// TIA Portal project "bary_callebaut" (V14)

(* hardware
DEVICE "S7-1200 station_1"  S7-1200 Station
   slot 0: "Rack_0"  S7-1200 Rack  Rack  V1.0
   slot 1: "PLC_1"  CPU 1214C DC/DC/DC  6ES7 214-1AG40-0XB0  V4.2
   slot 2: "DI 8/DQ 8x24VDC_1"  6ES7 223-1BH32-0XB0  V2.0
   slot 3: "SIWAREX WP231"  SIWAREX WP231  7MH4960-2AA01
DEVICE "GSD device_2"  GSD.Device.PN
   slot 0: "Rack"  Rack  V1.0
   slot 0: "danfoss-fc-series"  Danfoss FC PN  132B0348  V03.01.0
      slot 0: "Danfoss FC PN"  Danfoss FC PN
      slot 1: "Interface"  Interface
         slot 1: "Port 1"  Port 1
         slot 2: "Port 2"  Port 2
   slot 1: "PPO 6 - 4/4 Words, Danfoss Telegram 106_1"  PPO 6 - 4/4 Words, Danfoss Telegram 106
      slot 0: "Parameter Access Point"  Parameter Access Point
      slot 1: "PPO 6 - 4/4 Words, Danfoss Telegram 106"  PPO 6 - 4/4 Words, Danfoss Telegram 106
DEVICE "HMI"  TP700 Comfort
   slot 0: "HMI"  HMI  6AV2 124-0GC01-0AX0  13.0.1.0
   slot 1: "HMI_RT_2"  TP700 Comfort  6AV2 124-0GC01-0AX0  13.0.1.0
   slot 5: "HMI.IE_CP_1"  PROFINET Schnittstelle
      slot 1: "PROFINET Schnittstelle_1"  PROFINET Schnittstelle
         slot 1: "Port_1"  Port
         slot 2: "Port_2"  Port
   slot 7: "HMI.MPI/DP_CP_1"  MPI/DP Schnittstelle
DEVICE "HMI_1"  KTP700 Basic PN
   slot 0: "KTP700 Basic PN"  KTP700 Basic PN  6AV2 123-2GB03-0AX0  14.0.1.0
   slot 1: "HMI_RT_1"  KTP700 Basic PN  6AV2 123-2GB03-0AX0  14.0.1.0
   slot 5: "HMI_1.IE_CP_1"  PROFINET Interface  14.0.1.0
      slot 1: "PROFINET Interface_1"  PROFINET Interface
         slot 1: "Port_1"  Port
*)

// ===== PLC "PLC_1"  CPU 1214C DC/DC/DC =====
// protected blocks, not shown: "WP231PR"

VAR_GLOBAL   // PLC tag table "Default tag table"
   "Voltage_CPU_Ok" AT %I0.0 : Bool;   // Питание контрллера в номе
   "Voltage_DI_Ok" AT %I0.1 : Bool;   // Питание DI в норме
   "Voltage_DO_Ok" AT %I0.2 : Bool;   // Питание DO в норме
   "Voltage_24V_Ok" AT %I0.3 : Bool;   // Питание 24В в норме
   "Safety_Ok" AT %I0.4 : Bool;   // Безопасность в норме
   "Cold_tunnel_QF" AT %I0.5 : Bool;   // Защитный автомат холодный тунель
   "T1_QF" AT %I0.6 : Bool;   // Защитный автомат Т1
   "T2_QF" AT %I0.7 : Bool;   // Защитный автомат Т2
   "T3_QF" AT %I1.0 : Bool;   // Защитный автомат Т3
   "T2_Box_ready" AT %I1.1 : Bool;   // Датчик наличия коробки
   "T3_Box_ready" AT %I1.2 : Bool;   // Датчик наличия коробки
   "T4_Box_ready" AT %I1.3 : Bool;   // Датчик наличия коробки
   "Air_pressure_Ok" AT %I1.4 : Bool;   // Давление воздуха
   "FB_K1_Close" AT %I2.0 : Bool;   // Закрыто
   "FB_K2_Open" AT %I2.1 : Bool;   // Открыто
   "FB_K2_Close" AT %I2.2 : Bool;   // Закрыто
   "FB_K3_Open" AT %I2.3 : Bool;   // Открыто
   "FB_K3_Close" AT %I2.4 : Bool;   // Закрыто
   "T0_CMD" AT %Q0.0 : Bool;   // Вкл Т0
   "T1_CMD" AT %Q0.1 : Bool;   // Вкл Т1
   "T2_CMD" AT %Q0.2 : Bool;   // Вкл Т2
   "T3_CMD" AT %Q0.3 : Bool;   // Вкл Т3
   "K1_CMD" AT %Q0.4 : Bool;   // Вкл/выкл К1
   "K2_CMD" AT %Q0.5 : Bool;   // Вкл К2
   "K3_CMD" AT %Q0.6 : Bool;   // Вкл К3
   "Supply_allowed" AT %Q0.7 : Bool;   // Подача шоколада разрешена (отдаем другой системе)
   "Reset_safety" AT %Q2.0 : Bool;   // Сброс безопасности
   "Reset" AT %Q2.1 : Bool;   // Сброс
   "Green" AT %Q2.4 : Bool;   // Зеленый
   "Red" AT %Q2.5 : Bool;   // Красный
   "Blue" AT %Q2.6 : Bool;   // Синий
   "Orange" AT %Q2.7 : Bool;   // Оранжевый
   "Tag_1" AT %MW50 : Int;
   "Tag_2" AT %M100.0 : Bool;
END_VAR

VAR_GLOBAL   // PLC tag table "CF_tegs"
   "Status_word_input" AT %IW50 : Int;
   "MAV_input" AT %IW52 : Int;
   "Motor_torque_input" AT %IW54 : Int;
   "Digital_input" AT %IW56 : Int;
   "Control_word_output" AT %QW50 : Int;
   "Not_used_output" AT %QW54 : Int;
   "Reference_output" AT %QW52 : Int;
   "Not_used_output(1)" AT %QW56 : Int;
END_VAR

VAR_GLOBAL   // PLC tag table "Sys"
   "ON" AT %M2.0 : Bool;
   "OFF" AT %M2.1 : Bool;
   "pulse_01s" AT %M3.0 : Bool;
   "pulse_05s" AT %M3.1 : Bool;
   "pulse_1s" AT %M3.2 : Bool;
   "pulse_1m" AT %M3.3 : Bool;
   "pulse_1h" AT %M3.4 : Bool;
   "All_block" AT %M4.0 : Bool;
   "Reset_All" AT %M4.1 : Bool;
   "Sim_All" AT %M4.2 : Bool;
   "Global_Alm" AT %M4.3 : Bool;
   "ToAuto" AT %M4.4 : Bool;
   "ToHand" AT %M4.5 : Bool;
   "Any_Hand" AT %M5.0 : Bool;
   "DI_Hand" AT %M5.1 : Bool;
   "DO_Hand" AT %M5.2 : Bool;
   "AI_Hand" AT %M5.3 : Bool;
   "AO_Hand" AT %M5.4 : Bool;
   "M_Hand" AT %M5.5 : Bool;
   "V_Hand" AT %M5.6 : Bool;
   "X_Hand" AT %M5.7 : Bool;
   "System_Byte" AT %MB1 : Byte;
   "FirstScan" AT %M1.0 : Bool;
   "DiagStatusUpdate" AT %M1.1 : Bool;
   "AlwaysTRUE" AT %M1.2 : Bool;
   "AlwaysFALSE" AT %M1.3 : Bool;
   "Clock_Byte" AT %MB0 : Byte;
   "Clock_10Hz" AT %M0.0 : Bool;
   "Clock_5Hz" AT %M0.1 : Bool;
   "Clock_2.5Hz" AT %M0.2 : Bool;
   "Clock_2Hz" AT %M0.3 : Bool;
   "Clock_1.25Hz" AT %M0.4 : Bool;
   "Clock_1Hz" AT %M0.5 : Bool;
   "Clock_0.625Hz" AT %M0.6 : Bool;
   "Clock_0.5Hz" AT %M0.7 : Bool;
   "DI_Alm" AT %M6.0 : Bool;
   "DO_Alm" AT %M6.1 : Bool;
   "AI_Alm" AT %M6.2 : Bool;
   "AO_Alm" AT %M6.3 : Bool;
   "M_Alm" AT %M6.4 : Bool;
   "V_Alm" AT %M6.5 : Bool;
   "X_Alm" AT %M6.6 : Bool;
   "Any_Alm" AT %M6.7 : Bool;
   "W_Alm" AT %M7.0 : Bool;
   "RPD_Alm" AT %M7.1 : Bool;
   "I_Alm" AT %M7.2 : Bool;
   "O1_Alm" AT %M7.3 : Bool;
   "O2_Alm" AT %M7.4 : Bool;
   "VT_Alm" AT %M7.5 : Bool;
   "FStop" AT %M7.6 : Bool;
   "pulse_5s" AT %M3.5 : Bool;
   "Clock_5s" AT %M3.6 : Bool;
   "pos_1s" AT %M8.0 : Bool;
   "pos_05s" AT %M8.1 : Bool;
   "pos_01s" AT %M8.2 : Bool;
   "neg_01s" AT %M8.3 : Bool;
END_VAR

DATA_BLOCK "Logic_DB"   // DB4
{ S7_Optimized_Access := 'FALSE' }
VERSION : 0.1
// stored: InstanceOfName Logic
"Logic"
BEGIN
   T_reset_mem.SP := 10.0;
END_DATA_BLOCK

DATA_BLOCK "T4D4_DB"   // DB10
{ S7_Optimized_Access := 'FALSE' }
VERSION : 0.1
// stored: InstanceOfName T4D4
"T4D4"
BEGIN
   S2.One := 0.1;
   S2.SP := 5.0;
   S1.One := 0.1;
   S1.SP := 2.0;
END_DATA_BLOCK

DATA_BLOCK "T3V3W3_DB"   // DB11
{ S7_Optimized_Access := 'FALSE' }
VERSION : 0.1
// stored: InstanceOfName T3V3W3
"T3V3W3"
BEGIN
END_DATA_BLOCK

DATA_BLOCK "T2D2_DB"   // DB12
{ S7_Optimized_Access := 'FALSE' }
VERSION : 0.1
// stored: InstanceOfName T2D2
"T2D2"
BEGIN
END_DATA_BLOCK

DATA_BLOCK "T0T1_DB"   // DB13
{ S7_Optimized_Access := 'FALSE' }
VERSION : 0.1
// stored: InstanceOfName T0T1
"T0T1"
BEGIN
END_DATA_BLOCK

DATA_BLOCK "del_stat_mem_DB"   // DB14
{ S7_Optimized_Access := 'FALSE' }
VERSION : 0.1
// stored: InstanceOfName del_stat_mem
"del_stat_mem"
BEGIN
END_DATA_BLOCK

DATA_BLOCK "move_pn_DB"   // DB16
{ S7_Optimized_Access := 'FALSE' }
VERSION : 0.1
// stored: InstanceOfName move_pn
"move_pn"
BEGIN
END_DATA_BLOCK

DATA_BLOCK "Reset_st_DB"   // DB17
{ S7_Optimized_Access := 'FALSE' }
VERSION : 0.1
// stored: InstanceOfName Reset_st
"Reset_st"
BEGIN
END_DATA_BLOCK

DATA_BLOCK "Statistic_DB"   // DB19
{ S7_Optimized_Access := 'FALSE' }
VERSION : 0.1
// stored: InstanceOfName Statistic
"Statistic"
BEGIN
END_DATA_BLOCK

DATA_BLOCK "prepare_DB"   // DB20
{ S7_Optimized_Access := 'TRUE' }
VERSION : 0.1
// stored: InstanceOfName prepare
"prepare"
BEGIN
END_DATA_BLOCK

// folder: Modules

DATA_BLOCK "Profinet_FC280_DB"   // DB1
{ S7_Optimized_Access := 'FALSE' }
VERSION : 0.1
// stored: InstanceOfName Profinet_FC280
"Profinet_FC280"
BEGIN
END_DATA_BLOCK

DATA_BLOCK "Motors_DB"   // DB2
{ S7_Optimized_Access := 'FALSE' }
VERSION : 0.1
// stored: InstanceOfName Motors
"Motors"
BEGIN
END_DATA_BLOCK

DATA_BLOCK "Valves_DB"   // DB3
{ S7_Optimized_Access := 'FALSE' }
VERSION : 0.1
// stored: InstanceOfName Valves
"Valves"
BEGIN
END_DATA_BLOCK

DATA_BLOCK "DRV_CF_DB"   // DB5
{ S7_Optimized_Access := 'FALSE' }
VERSION : 0.1
// stored: InstanceOfName DRV_CF
"DRV_CF"
BEGIN
END_DATA_BLOCK

DATA_BLOCK "DOx_DB"   // DB6
{ S7_Optimized_Access := 'FALSE' }
VERSION : 0.1
// stored: InstanceOfName DOx
"DOx"
BEGIN
END_DATA_BLOCK

DATA_BLOCK "AOx_DB"   // DB8
{ S7_Optimized_Access := 'FALSE' }
VERSION : 0.1
// stored: InstanceOfName AOx
"AOx"
BEGIN
END_DATA_BLOCK

DATA_BLOCK "DIx_DB"   // DB9
{ S7_Optimized_Access := 'FALSE' }
VERSION : 0.1
// stored: InstanceOfName DIx
"DIx"
BEGIN
END_DATA_BLOCK

// folder: System blocks/Program resources

DATA_BLOCK "T_Reset"   // DB7
{ S7_Optimized_Access := 'TRUE' }
AUTHOR : Simatic
FAMILY : IEC
NAME : IEC_TMR
VERSION : 1.0
// stored: InstanceOfName IEC_TIMER
"IEC_TIMER"
BEGIN
END_DATA_BLOCK

DATA_BLOCK "clock_5s_ON"   // DB507
{ S7_Optimized_Access := 'TRUE' }
AUTHOR : Simatic
FAMILY : IEC
NAME : IEC_TMR
VERSION : 1.0
// stored: InstanceOfName IEC_TIMER
"IEC_TIMER"
BEGIN
END_DATA_BLOCK

DATA_BLOCK "clock_5s_OFF"   // DB508
{ S7_Optimized_Access := 'TRUE' }
AUTHOR : Simatic
FAMILY : IEC
NAME : IEC_TMR
VERSION : 1.0
// stored: InstanceOfName IEC_TIMER
"IEC_TIMER"
BEGIN
END_DATA_BLOCK

// folder: db_flash

DATA_BLOCK "data"   // DB15
{ S7_Optimized_Access := 'FALSE' }
VERSION : 0.1
   VAR
      newName : String := 'newlog';
      "name" : String := 'log';
      logID : DWord;
      logHeader : String := 'count,weight';
      myData : Struct
         number : Int;
         weight : Real;
      END_STRUCT;
      executeCreate : Bool;
      crateDone : Bool;
      createBusy : Bool;
      createError : Bool;
      createStatus : Word;
      createStatusMem : Word;
      dlogCreated : Bool;
   END_VAR
BEGIN
END_DATA_BLOCK

DATA_BLOCK "logW"   // DB21
{ S7_Optimized_Access := 'TRUE' }
VERSION : 0.1
   VAR
      executeWrite : Bool;
      count : Int;
      scaledTemp : Real;
      scaledPressure : Real;
      writeDone : Bool;
      writeBusy : Bool;
      writeError : Bool;
      writeFullStatus : Word;
      closeDone : Bool;
      closeBusy : Bool;
      closeError : Bool;
      closeStatus : Word;
      executeOpen : Bool;
      openDone : Bool;
      openBusy : Bool;
      openError : Bool;
      openStatus : Word;
      executeNewFile : Bool;
      fileDone : Bool;
      fileBusy : Bool;
      fileError : Bool;
      fileStatus : Word;
   END_VAR
BEGIN
END_DATA_BLOCK

DATA_BLOCK "logFB"   // DB22
{ S7_Optimized_Access := 'TRUE' }
VERSION : 0.1
BEGIN
END_DATA_BLOCK

// folder: statistic

DATA_BLOCK "bd"   // DB18
{ S7_Optimized_Access := 'FALSE' }
VERSION : 0.1
   VAR
      weight_box : Array[1..3000] of Real;
   END_VAR
BEGIN
   weight_box[1] := 0.0;
   weight_box[2] := 0.0;
   weight_box[3] := 0.0;
   weight_box[4] := 0.0;
   weight_box[5] := 0.0;
   weight_box[6] := 0.0;
   weight_box[7] := 0.0;
   weight_box[8] := 0.0;
   weight_box[9] := 0.0;
   weight_box[10] := 0.0;
   weight_box[11] := 0.0;
   weight_box[12] := 0.0;
   weight_box[13] := 0.0;
   weight_box[14] := 0.0;
   weight_box[15] := 0.0;
   weight_box[16] := 0.0;
   weight_box[17] := 0.0;
   weight_box[18] := 0.0;
   weight_box[19] := 0.0;
   weight_box[20] := 0.0;
   weight_box[21] := 0.0;
   weight_box[22] := 0.0;
   weight_box[23] := 0.0;
   weight_box[24] := 0.0;
   weight_box[25] := 0.0;
   weight_box[26] := 0.0;
   weight_box[27] := 0.0;
   weight_box[28] := 0.0;
   weight_box[29] := 0.0;
   weight_box[30] := 0.0;
   weight_box[31] := 0.0;
   weight_box[32] := 0.0;
   weight_box[33] := 0.0;
   weight_box[34] := 0.0;
   weight_box[35] := 0.0;
   weight_box[36] := 0.0;
   weight_box[37] := 0.0;
   weight_box[38] := 0.0;
   weight_box[39] := 0.0;
   weight_box[40] := 0.0;
   weight_box[41] := 0.0;
   weight_box[42] := 0.0;
   weight_box[43] := 0.0;
   weight_box[44] := 0.0;
   weight_box[45] := 0.0;
   weight_box[46] := 0.0;
   weight_box[47] := 0.0;
   weight_box[48] := 0.0;
   weight_box[49] := 0.0;
   weight_box[50] := 0.0;
   weight_box[51] := 0.0;
   weight_box[52] := 0.0;
   weight_box[53] := 0.0;
   weight_box[54] := 0.0;
   weight_box[55] := 0.0;
   weight_box[56] := 0.0;
   weight_box[57] := 0.0;
   weight_box[58] := 0.0;
   weight_box[59] := 0.0;
   weight_box[60] := 0.0;
   weight_box[61] := 0.0;
   weight_box[62] := 0.0;
   weight_box[63] := 0.0;
   weight_box[64] := 0.0;
   weight_box[65] := 0.0;
   weight_box[66] := 0.0;
   weight_box[67] := 0.0;
   weight_box[68] := 0.0;
   weight_box[69] := 0.0;
   weight_box[70] := 0.0;
   weight_box[71] := 0.0;
   weight_box[72] := 0.0;
   weight_box[73] := 0.0;
   weight_box[74] := 0.0;
   weight_box[75] := 0.0;
   weight_box[76] := 0.0;
   weight_box[77] := 0.0;
   weight_box[78] := 0.0;
   weight_box[79] := 0.0;
   weight_box[80] := 0.0;
   weight_box[81] := 0.0;
   weight_box[82] := 0.0;
   weight_box[83] := 0.0;
   weight_box[84] := 0.0;
   weight_box[85] := 0.0;
   weight_box[86] := 0.0;
   weight_box[87] := 0.0;
   weight_box[88] := 0.0;
   weight_box[89] := 0.0;
   weight_box[90] := 0.0;
   weight_box[91] := 0.0;
   weight_box[92] := 0.0;
   weight_box[93] := 0.0;
   weight_box[94] := 0.0;
   weight_box[95] := 0.0;
   weight_box[96] := 0.0;
   weight_box[97] := 0.0;
   weight_box[98] := 0.0;
   weight_box[99] := 0.0;
   weight_box[100] := 0.0;
   weight_box[101] := 0.0;
   weight_box[102] := 0.0;
   weight_box[103] := 0.0;
   weight_box[104] := 0.0;
   weight_box[105] := 0.0;
   weight_box[106] := 0.0;
   weight_box[107] := 0.0;
   weight_box[108] := 0.0;
   weight_box[109] := 0.0;
   weight_box[110] := 0.0;
   weight_box[111] := 0.0;
   weight_box[112] := 0.0;
   weight_box[113] := 0.0;
   weight_box[114] := 0.0;
   weight_box[115] := 0.0;
   weight_box[116] := 0.0;
   weight_box[117] := 0.0;
   weight_box[118] := 0.0;
   weight_box[119] := 0.0;
   weight_box[120] := 0.0;
   weight_box[121] := 0.0;
   weight_box[122] := 0.0;
   weight_box[123] := 0.0;
   weight_box[124] := 0.0;
   weight_box[125] := 0.0;
   weight_box[126] := 0.0;
   weight_box[127] := 0.0;
   weight_box[128] := 0.0;
   weight_box[129] := 0.0;
   weight_box[130] := 0.0;
   weight_box[131] := 0.0;
   weight_box[132] := 0.0;
   weight_box[133] := 0.0;
   weight_box[134] := 0.0;
   weight_box[135] := 0.0;
   weight_box[136] := 0.0;
   weight_box[137] := 0.0;
   weight_box[138] := 0.0;
   weight_box[139] := 0.0;
   weight_box[140] := 0.0;
   weight_box[141] := 0.0;
   weight_box[142] := 0.0;
   weight_box[143] := 0.0;
   weight_box[144] := 0.0;
   weight_box[145] := 0.0;
   weight_box[146] := 0.0;
   weight_box[147] := 0.0;
   weight_box[148] := 0.0;
   weight_box[149] := 0.0;
   weight_box[150] := 0.0;
   weight_box[151] := 0.0;
   weight_box[152] := 0.0;
   weight_box[153] := 0.0;
   weight_box[154] := 0.0;
   weight_box[155] := 0.0;
   weight_box[156] := 0.0;
   weight_box[157] := 0.0;
   weight_box[158] := 0.0;
   weight_box[159] := 0.0;
   weight_box[160] := 0.0;
   weight_box[161] := 0.0;
   weight_box[162] := 0.0;
   weight_box[163] := 0.0;
   weight_box[164] := 0.0;
   weight_box[165] := 0.0;
   weight_box[166] := 0.0;
   weight_box[167] := 0.0;
   weight_box[168] := 0.0;
   weight_box[169] := 0.0;
   weight_box[170] := 0.0;
   weight_box[171] := 0.0;
   weight_box[172] := 0.0;
   weight_box[173] := 0.0;
   weight_box[174] := 0.0;
   weight_box[175] := 0.0;
   weight_box[176] := 0.0;
   weight_box[177] := 0.0;
   weight_box[178] := 0.0;
   weight_box[179] := 0.0;
   weight_box[180] := 0.0;
   weight_box[181] := 0.0;
   weight_box[182] := 0.0;
   weight_box[183] := 0.0;
   weight_box[184] := 0.0;
   weight_box[185] := 0.0;
   weight_box[186] := 0.0;
   weight_box[187] := 0.0;
   weight_box[188] := 0.0;
   weight_box[189] := 0.0;
   weight_box[190] := 0.0;
   weight_box[191] := 0.0;
   weight_box[192] := 0.0;
   weight_box[193] := 0.0;
   weight_box[194] := 0.0;
   weight_box[195] := 0.0;
   weight_box[196] := 0.0;
   weight_box[197] := 0.0;
   weight_box[198] := 0.0;
   weight_box[199] := 0.0;
   weight_box[200] := 0.0;
   weight_box[201] := 0.0;
   weight_box[202] := 0.0;
   weight_box[203] := 0.0;
   weight_box[204] := 0.0;
   weight_box[205] := 0.0;
   weight_box[206] := 0.0;
   weight_box[207] := 0.0;
   weight_box[208] := 0.0;
   weight_box[209] := 0.0;
   weight_box[210] := 0.0;
   weight_box[211] := 0.0;
   weight_box[212] := 0.0;
   weight_box[213] := 0.0;
   weight_box[214] := 0.0;
   weight_box[215] := 0.0;
   weight_box[216] := 0.0;
   weight_box[217] := 0.0;
   weight_box[218] := 0.0;
   weight_box[219] := 0.0;
   weight_box[220] := 0.0;
   weight_box[221] := 0.0;
   weight_box[222] := 0.0;
   weight_box[223] := 0.0;
   weight_box[224] := 0.0;
   weight_box[225] := 0.0;
   weight_box[226] := 0.0;
   weight_box[227] := 0.0;
   weight_box[228] := 0.0;
   weight_box[229] := 0.0;
   weight_box[230] := 0.0;
   weight_box[231] := 0.0;
   weight_box[232] := 0.0;
   weight_box[233] := 0.0;
   weight_box[234] := 0.0;
   weight_box[235] := 0.0;
   weight_box[236] := 0.0;
   weight_box[237] := 0.0;
   weight_box[238] := 0.0;
   weight_box[239] := 0.0;
   weight_box[240] := 0.0;
   weight_box[241] := 0.0;
   weight_box[242] := 0.0;
   weight_box[243] := 0.0;
   weight_box[244] := 0.0;
   weight_box[245] := 0.0;
   weight_box[246] := 0.0;
   weight_box[247] := 0.0;
   weight_box[248] := 0.0;
   weight_box[249] := 0.0;
   weight_box[250] := 0.0;
   weight_box[251] := 0.0;
   weight_box[252] := 0.0;
   weight_box[253] := 0.0;
   weight_box[254] := 0.0;
   weight_box[255] := 0.0;
   weight_box[256] := 0.0;
   weight_box[257] := 0.0;
   weight_box[258] := 0.0;
   weight_box[259] := 0.0;
   weight_box[260] := 0.0;
   weight_box[261] := 0.0;
   weight_box[262] := 0.0;
   weight_box[263] := 0.0;
   weight_box[264] := 0.0;
   weight_box[265] := 0.0;
   weight_box[266] := 0.0;
   weight_box[267] := 0.0;
   weight_box[268] := 0.0;
   weight_box[269] := 0.0;
   weight_box[270] := 0.0;
   weight_box[271] := 0.0;
   weight_box[272] := 0.0;
   weight_box[273] := 0.0;
   weight_box[274] := 0.0;
   weight_box[275] := 0.0;
   weight_box[276] := 0.0;
   weight_box[277] := 0.0;
   weight_box[278] := 0.0;
   weight_box[279] := 0.0;
   weight_box[280] := 0.0;
   weight_box[281] := 0.0;
   weight_box[282] := 0.0;
   weight_box[283] := 0.0;
   weight_box[284] := 0.0;
   weight_box[285] := 0.0;
   weight_box[286] := 0.0;
   weight_box[287] := 0.0;
   weight_box[288] := 0.0;
   weight_box[289] := 0.0;
   weight_box[290] := 0.0;
   weight_box[291] := 0.0;
   weight_box[292] := 0.0;
   weight_box[293] := 0.0;
   weight_box[294] := 0.0;
   weight_box[295] := 0.0;
   weight_box[296] := 0.0;
   weight_box[297] := 0.0;
   weight_box[298] := 0.0;
   weight_box[299] := 0.0;
   weight_box[300] := 0.0;
   weight_box[301] := 0.0;
   weight_box[302] := 0.0;
   weight_box[303] := 0.0;
   weight_box[304] := 0.0;
   weight_box[305] := 0.0;
   weight_box[306] := 0.0;
   weight_box[307] := 0.0;
   weight_box[308] := 0.0;
   weight_box[309] := 0.0;
   weight_box[310] := 0.0;
   weight_box[311] := 0.0;
   weight_box[312] := 0.0;
   weight_box[313] := 0.0;
   weight_box[314] := 0.0;
   weight_box[315] := 0.0;
   weight_box[316] := 0.0;
   weight_box[317] := 0.0;
   weight_box[318] := 0.0;
   weight_box[319] := 0.0;
   weight_box[320] := 0.0;
   weight_box[321] := 0.0;
   weight_box[322] := 0.0;
   weight_box[323] := 0.0;
   weight_box[324] := 0.0;
   weight_box[325] := 0.0;
   weight_box[326] := 0.0;
   weight_box[327] := 0.0;
   weight_box[328] := 0.0;
   weight_box[329] := 0.0;
   weight_box[330] := 0.0;
   weight_box[331] := 0.0;
   weight_box[332] := 0.0;
   weight_box[333] := 0.0;
   weight_box[334] := 0.0;
   weight_box[335] := 0.0;
   weight_box[336] := 0.0;
   weight_box[337] := 0.0;
   weight_box[338] := 0.0;
   weight_box[339] := 0.0;
   weight_box[340] := 0.0;
   weight_box[341] := 0.0;
   weight_box[342] := 0.0;
   weight_box[343] := 0.0;
   weight_box[344] := 0.0;
   weight_box[345] := 0.0;
   weight_box[346] := 0.0;
   weight_box[347] := 0.0;
   weight_box[348] := 0.0;
   weight_box[349] := 0.0;
   weight_box[350] := 0.0;
   weight_box[351] := 0.0;
   weight_box[352] := 0.0;
   weight_box[353] := 0.0;
   weight_box[354] := 0.0;
   weight_box[355] := 0.0;
   weight_box[356] := 0.0;
   weight_box[357] := 0.0;
   weight_box[358] := 0.0;
   weight_box[359] := 0.0;
   weight_box[360] := 0.0;
   weight_box[361] := 0.0;
   weight_box[362] := 0.0;
   weight_box[363] := 0.0;
   weight_box[364] := 0.0;
   weight_box[365] := 0.0;
   weight_box[366] := 0.0;
   weight_box[367] := 0.0;
   weight_box[368] := 0.0;
   weight_box[369] := 0.0;
   weight_box[370] := 0.0;
   weight_box[371] := 0.0;
   weight_box[372] := 0.0;
   weight_box[373] := 0.0;
   weight_box[374] := 0.0;
   weight_box[375] := 0.0;
   weight_box[376] := 0.0;
   weight_box[377] := 0.0;
   weight_box[378] := 0.0;
   weight_box[379] := 0.0;
   weight_box[380] := 0.0;
   weight_box[381] := 0.0;
   weight_box[382] := 0.0;
   weight_box[383] := 0.0;
   weight_box[384] := 0.0;
   weight_box[385] := 0.0;
   weight_box[386] := 0.0;
   weight_box[387] := 0.0;
   weight_box[388] := 0.0;
   weight_box[389] := 0.0;
   weight_box[390] := 0.0;
   weight_box[391] := 0.0;
   weight_box[392] := 0.0;
   weight_box[393] := 0.0;
   weight_box[394] := 0.0;
   weight_box[395] := 0.0;
   weight_box[396] := 0.0;
   weight_box[397] := 0.0;
   weight_box[398] := 0.0;
   weight_box[399] := 0.0;
   weight_box[400] := 0.0;
   weight_box[401] := 0.0;
   weight_box[402] := 0.0;
   weight_box[403] := 0.0;
   weight_box[404] := 0.0;
   weight_box[405] := 0.0;
   weight_box[406] := 0.0;
   weight_box[407] := 0.0;
   weight_box[408] := 0.0;
   weight_box[409] := 0.0;
   weight_box[410] := 0.0;
   weight_box[411] := 0.0;
   weight_box[412] := 0.0;
   weight_box[413] := 0.0;
   weight_box[414] := 0.0;
   weight_box[415] := 0.0;
   weight_box[416] := 0.0;
   weight_box[417] := 0.0;
   weight_box[418] := 0.0;
   weight_box[419] := 0.0;
   weight_box[420] := 0.0;
   weight_box[421] := 0.0;
   weight_box[422] := 0.0;
   weight_box[423] := 0.0;
   weight_box[424] := 0.0;
   weight_box[425] := 0.0;
   weight_box[426] := 0.0;
   weight_box[427] := 0.0;
   weight_box[428] := 0.0;
   weight_box[429] := 0.0;
   weight_box[430] := 0.0;
   weight_box[431] := 0.0;
   weight_box[432] := 0.0;
   weight_box[433] := 0.0;
   weight_box[434] := 0.0;
   weight_box[435] := 0.0;
   weight_box[436] := 0.0;
   weight_box[437] := 0.0;
   weight_box[438] := 0.0;
   weight_box[439] := 0.0;
   weight_box[440] := 0.0;
   weight_box[441] := 0.0;
   weight_box[442] := 0.0;
   weight_box[443] := 0.0;
   weight_box[444] := 0.0;
   weight_box[445] := 0.0;
   weight_box[446] := 0.0;
   weight_box[447] := 0.0;
   weight_box[448] := 0.0;
   weight_box[449] := 0.0;
   weight_box[450] := 0.0;
   weight_box[451] := 0.0;
   weight_box[452] := 0.0;
   weight_box[453] := 0.0;
   weight_box[454] := 0.0;
   weight_box[455] := 0.0;
   weight_box[456] := 0.0;
   weight_box[457] := 0.0;
   weight_box[458] := 0.0;
   weight_box[459] := 0.0;
   weight_box[460] := 0.0;
   weight_box[461] := 0.0;
   weight_box[462] := 0.0;
   weight_box[463] := 0.0;
   weight_box[464] := 0.0;
   weight_box[465] := 0.0;
   weight_box[466] := 0.0;
   weight_box[467] := 0.0;
   weight_box[468] := 0.0;
   weight_box[469] := 0.0;
   weight_box[470] := 0.0;
   weight_box[471] := 0.0;
   weight_box[472] := 0.0;
   weight_box[473] := 0.0;
   weight_box[474] := 0.0;
   weight_box[475] := 0.0;
   weight_box[476] := 0.0;
   weight_box[477] := 0.0;
   weight_box[478] := 0.0;
   weight_box[479] := 0.0;
   weight_box[480] := 0.0;
   weight_box[481] := 0.0;
   weight_box[482] := 0.0;
   weight_box[483] := 0.0;
   weight_box[484] := 0.0;
   weight_box[485] := 0.0;
   weight_box[486] := 0.0;
   weight_box[487] := 0.0;
   weight_box[488] := 0.0;
   weight_box[489] := 0.0;
   weight_box[490] := 0.0;
   weight_box[491] := 0.0;
   weight_box[492] := 0.0;
   weight_box[493] := 0.0;
   weight_box[494] := 0.0;
   weight_box[495] := 0.0;
   weight_box[496] := 0.0;
   weight_box[497] := 0.0;
   weight_box[498] := 0.0;
   weight_box[499] := 0.0;
   weight_box[500] := 0.0;
   weight_box[501] := 0.0;
   weight_box[502] := 0.0;
   weight_box[503] := 0.0;
   weight_box[504] := 0.0;
   weight_box[505] := 0.0;
   weight_box[506] := 0.0;
   weight_box[507] := 0.0;
   weight_box[508] := 0.0;
   weight_box[509] := 0.0;
   weight_box[510] := 0.0;
   weight_box[511] := 0.0;
   weight_box[512] := 0.0;
   weight_box[513] := 0.0;
   weight_box[514] := 0.0;
   weight_box[515] := 0.0;
   weight_box[516] := 0.0;
   weight_box[517] := 0.0;
   weight_box[518] := 0.0;
   weight_box[519] := 0.0;
   weight_box[520] := 0.0;
   weight_box[521] := 0.0;
   weight_box[522] := 0.0;
   weight_box[523] := 0.0;
   weight_box[524] := 0.0;
   weight_box[525] := 0.0;
   weight_box[526] := 0.0;
   weight_box[527] := 0.0;
   weight_box[528] := 0.0;
   weight_box[529] := 0.0;
   weight_box[530] := 0.0;
   weight_box[531] := 0.0;
   weight_box[532] := 0.0;
   weight_box[533] := 0.0;
   weight_box[534] := 0.0;
   weight_box[535] := 0.0;
   weight_box[536] := 0.0;
   weight_box[537] := 0.0;
   weight_box[538] := 0.0;
   weight_box[539] := 0.0;
   weight_box[540] := 0.0;
   weight_box[541] := 0.0;
   weight_box[542] := 0.0;
   weight_box[543] := 0.0;
   weight_box[544] := 0.0;
   weight_box[545] := 0.0;
   weight_box[546] := 0.0;
   weight_box[547] := 0.0;
   weight_box[548] := 0.0;
   weight_box[549] := 0.0;
   weight_box[550] := 0.0;
   weight_box[551] := 0.0;
   weight_box[552] := 0.0;
   weight_box[553] := 0.0;
   weight_box[554] := 0.0;
   weight_box[555] := 0.0;
   weight_box[556] := 0.0;
   weight_box[557] := 0.0;
   weight_box[558] := 0.0;
   weight_box[559] := 0.0;
   weight_box[560] := 0.0;
   weight_box[561] := 0.0;
   weight_box[562] := 0.0;
   weight_box[563] := 0.0;
   weight_box[564] := 0.0;
   weight_box[565] := 0.0;
   weight_box[566] := 0.0;
   weight_box[567] := 0.0;
   weight_box[568] := 0.0;
   weight_box[569] := 0.0;
   weight_box[570] := 0.0;
   weight_box[571] := 0.0;
   weight_box[572] := 0.0;
   weight_box[573] := 0.0;
   weight_box[574] := 0.0;
   weight_box[575] := 0.0;
   weight_box[576] := 0.0;
   weight_box[577] := 0.0;
   weight_box[578] := 0.0;
   weight_box[579] := 0.0;
   weight_box[580] := 0.0;
   weight_box[581] := 0.0;
   weight_box[582] := 0.0;
   weight_box[583] := 0.0;
   weight_box[584] := 0.0;
   weight_box[585] := 0.0;
   weight_box[586] := 0.0;
   weight_box[587] := 0.0;
   weight_box[588] := 0.0;
   weight_box[589] := 0.0;
   weight_box[590] := 0.0;
   weight_box[591] := 0.0;
   weight_box[592] := 0.0;
   weight_box[593] := 0.0;
   weight_box[594] := 0.0;
   weight_box[595] := 0.0;
   weight_box[596] := 0.0;
   weight_box[597] := 0.0;
   weight_box[598] := 0.0;
   weight_box[599] := 0.0;
   weight_box[600] := 0.0;
   weight_box[601] := 0.0;
   weight_box[602] := 0.0;
   weight_box[603] := 0.0;
   weight_box[604] := 0.0;
   weight_box[605] := 0.0;
   weight_box[606] := 0.0;
   weight_box[607] := 0.0;
   weight_box[608] := 0.0;
   weight_box[609] := 0.0;
   weight_box[610] := 0.0;
   weight_box[611] := 0.0;
   weight_box[612] := 0.0;
   weight_box[613] := 0.0;
   weight_box[614] := 0.0;
   weight_box[615] := 0.0;
   weight_box[616] := 0.0;
   weight_box[617] := 0.0;
   weight_box[618] := 0.0;
   weight_box[619] := 0.0;
   weight_box[620] := 0.0;
   weight_box[621] := 0.0;
   weight_box[622] := 0.0;
   weight_box[623] := 0.0;
   weight_box[624] := 0.0;
   weight_box[625] := 0.0;
   weight_box[626] := 0.0;
   weight_box[627] := 0.0;
   weight_box[628] := 0.0;
   weight_box[629] := 0.0;
   weight_box[630] := 0.0;
   weight_box[631] := 0.0;
   weight_box[632] := 0.0;
   weight_box[633] := 0.0;
   weight_box[634] := 0.0;
   weight_box[635] := 0.0;
   weight_box[636] := 0.0;
   weight_box[637] := 0.0;
   weight_box[638] := 0.0;
   weight_box[639] := 0.0;
   weight_box[640] := 0.0;
   weight_box[641] := 0.0;
   weight_box[642] := 0.0;
   weight_box[643] := 0.0;
   weight_box[644] := 0.0;
   weight_box[645] := 0.0;
   weight_box[646] := 0.0;
   weight_box[647] := 0.0;
   weight_box[648] := 0.0;
   weight_box[649] := 0.0;
   weight_box[650] := 0.0;
   weight_box[651] := 0.0;
   weight_box[652] := 0.0;
   weight_box[653] := 0.0;
   weight_box[654] := 0.0;
   weight_box[655] := 0.0;
   weight_box[656] := 0.0;
   weight_box[657] := 0.0;
   weight_box[658] := 0.0;
   weight_box[659] := 0.0;
   weight_box[660] := 0.0;
   weight_box[661] := 0.0;
   weight_box[662] := 0.0;
   weight_box[663] := 0.0;
   weight_box[664] := 0.0;
   weight_box[665] := 0.0;
   weight_box[666] := 0.0;
   weight_box[667] := 0.0;
   weight_box[668] := 0.0;
   weight_box[669] := 0.0;
   weight_box[670] := 0.0;
   weight_box[671] := 0.0;
   weight_box[672] := 0.0;
   weight_box[673] := 0.0;
   weight_box[674] := 0.0;
   weight_box[675] := 0.0;
   weight_box[676] := 0.0;
   weight_box[677] := 0.0;
   weight_box[678] := 0.0;
   weight_box[679] := 0.0;
   weight_box[680] := 0.0;
   weight_box[681] := 0.0;
   weight_box[682] := 0.0;
   weight_box[683] := 0.0;
   weight_box[684] := 0.0;
   weight_box[685] := 0.0;
   weight_box[686] := 0.0;
   weight_box[687] := 0.0;
   weight_box[688] := 0.0;
   weight_box[689] := 0.0;
   weight_box[690] := 0.0;
   weight_box[691] := 0.0;
   weight_box[692] := 0.0;
   weight_box[693] := 0.0;
   weight_box[694] := 0.0;
   weight_box[695] := 0.0;
   weight_box[696] := 0.0;
   weight_box[697] := 0.0;
   weight_box[698] := 0.0;
   weight_box[699] := 0.0;
   weight_box[700] := 0.0;
   weight_box[701] := 0.0;
   weight_box[702] := 0.0;
   weight_box[703] := 0.0;
   weight_box[704] := 0.0;
   weight_box[705] := 0.0;
   weight_box[706] := 0.0;
   weight_box[707] := 0.0;
   weight_box[708] := 0.0;
   weight_box[709] := 0.0;
   weight_box[710] := 0.0;
   weight_box[711] := 0.0;
   weight_box[712] := 0.0;
   weight_box[713] := 0.0;
   weight_box[714] := 0.0;
   weight_box[715] := 0.0;
   weight_box[716] := 0.0;
   weight_box[717] := 0.0;
   weight_box[718] := 0.0;
   weight_box[719] := 0.0;
   weight_box[720] := 0.0;
   weight_box[721] := 0.0;
   weight_box[722] := 0.0;
   weight_box[723] := 0.0;
   weight_box[724] := 0.0;
   weight_box[725] := 0.0;
   weight_box[726] := 0.0;
   weight_box[727] := 0.0;
   weight_box[728] := 0.0;
   weight_box[729] := 0.0;
   weight_box[730] := 0.0;
   weight_box[731] := 0.0;
   weight_box[732] := 0.0;
   weight_box[733] := 0.0;
   weight_box[734] := 0.0;
   weight_box[735] := 0.0;
   weight_box[736] := 0.0;
   weight_box[737] := 0.0;
   weight_box[738] := 0.0;
   weight_box[739] := 0.0;
   weight_box[740] := 0.0;
   weight_box[741] := 0.0;
   weight_box[742] := 0.0;
   weight_box[743] := 0.0;
   weight_box[744] := 0.0;
   weight_box[745] := 0.0;
   weight_box[746] := 0.0;
   weight_box[747] := 0.0;
   weight_box[748] := 0.0;
   weight_box[749] := 0.0;
   weight_box[750] := 0.0;
   weight_box[751] := 0.0;
   weight_box[752] := 0.0;
   weight_box[753] := 0.0;
   weight_box[754] := 0.0;
   weight_box[755] := 0.0;
   weight_box[756] := 0.0;
   weight_box[757] := 0.0;
   weight_box[758] := 0.0;
   weight_box[759] := 0.0;
   weight_box[760] := 0.0;
   weight_box[761] := 0.0;
   weight_box[762] := 0.0;
   weight_box[763] := 0.0;
   weight_box[764] := 0.0;
   weight_box[765] := 0.0;
   weight_box[766] := 0.0;
   weight_box[767] := 0.0;
   weight_box[768] := 0.0;
   weight_box[769] := 0.0;
   weight_box[770] := 0.0;
   weight_box[771] := 0.0;
   weight_box[772] := 0.0;
   weight_box[773] := 0.0;
   weight_box[774] := 0.0;
   weight_box[775] := 0.0;
   weight_box[776] := 0.0;
   weight_box[777] := 0.0;
   weight_box[778] := 0.0;
   weight_box[779] := 0.0;
   weight_box[780] := 0.0;
   weight_box[781] := 0.0;
   weight_box[782] := 0.0;
   weight_box[783] := 0.0;
   weight_box[784] := 0.0;
   weight_box[785] := 0.0;
   weight_box[786] := 0.0;
   weight_box[787] := 0.0;
   weight_box[788] := 0.0;
   weight_box[789] := 0.0;
   weight_box[790] := 0.0;
   weight_box[791] := 0.0;
   weight_box[792] := 0.0;
   weight_box[793] := 0.0;
   weight_box[794] := 0.0;
   weight_box[795] := 0.0;
   weight_box[796] := 0.0;
   weight_box[797] := 0.0;
   weight_box[798] := 0.0;
   weight_box[799] := 0.0;
   weight_box[800] := 0.0;
   weight_box[801] := 0.0;
   weight_box[802] := 0.0;
   weight_box[803] := 0.0;
   weight_box[804] := 0.0;
   weight_box[805] := 0.0;
   weight_box[806] := 0.0;
   weight_box[807] := 0.0;
   weight_box[808] := 0.0;
   weight_box[809] := 0.0;
   weight_box[810] := 0.0;
   weight_box[811] := 0.0;
   weight_box[812] := 0.0;
   weight_box[813] := 0.0;
   weight_box[814] := 0.0;
   weight_box[815] := 0.0;
   weight_box[816] := 0.0;
   weight_box[817] := 0.0;
   weight_box[818] := 0.0;
   weight_box[819] := 0.0;
   weight_box[820] := 0.0;
   weight_box[821] := 0.0;
   weight_box[822] := 0.0;
   weight_box[823] := 0.0;
   weight_box[824] := 0.0;
   weight_box[825] := 0.0;
   weight_box[826] := 0.0;
   weight_box[827] := 0.0;
   weight_box[828] := 0.0;
   weight_box[829] := 0.0;
   weight_box[830] := 0.0;
   weight_box[831] := 0.0;
   weight_box[832] := 0.0;
   weight_box[833] := 0.0;
   weight_box[834] := 0.0;
   weight_box[835] := 0.0;
   weight_box[836] := 0.0;
   weight_box[837] := 0.0;
   weight_box[838] := 0.0;
   weight_box[839] := 0.0;
   weight_box[840] := 0.0;
   weight_box[841] := 0.0;
   weight_box[842] := 0.0;
   weight_box[843] := 0.0;
   weight_box[844] := 0.0;
   weight_box[845] := 0.0;
   weight_box[846] := 0.0;
   weight_box[847] := 0.0;
   weight_box[848] := 0.0;
   weight_box[849] := 0.0;
   weight_box[850] := 0.0;
   weight_box[851] := 0.0;
   weight_box[852] := 0.0;
   weight_box[853] := 0.0;
   weight_box[854] := 0.0;
   weight_box[855] := 0.0;
   weight_box[856] := 0.0;
   weight_box[857] := 0.0;
   weight_box[858] := 0.0;
   weight_box[859] := 0.0;
   weight_box[860] := 0.0;
   weight_box[861] := 0.0;
   weight_box[862] := 0.0;
   weight_box[863] := 0.0;
   weight_box[864] := 0.0;
   weight_box[865] := 0.0;
   weight_box[866] := 0.0;
   weight_box[867] := 0.0;
   weight_box[868] := 0.0;
   weight_box[869] := 0.0;
   weight_box[870] := 0.0;
   weight_box[871] := 0.0;
   weight_box[872] := 0.0;
   weight_box[873] := 0.0;
   weight_box[874] := 0.0;
   weight_box[875] := 0.0;
   weight_box[876] := 0.0;
   weight_box[877] := 0.0;
   weight_box[878] := 0.0;
   weight_box[879] := 0.0;
   weight_box[880] := 0.0;
   weight_box[881] := 0.0;
   weight_box[882] := 0.0;
   weight_box[883] := 0.0;
   weight_box[884] := 0.0;
   weight_box[885] := 0.0;
   weight_box[886] := 0.0;
   weight_box[887] := 0.0;
   weight_box[888] := 0.0;
   weight_box[889] := 0.0;
   weight_box[890] := 0.0;
   weight_box[891] := 0.0;
   weight_box[892] := 0.0;
   weight_box[893] := 0.0;
   weight_box[894] := 0.0;
   weight_box[895] := 0.0;
   weight_box[896] := 0.0;
   weight_box[897] := 0.0;
   weight_box[898] := 0.0;
   weight_box[899] := 0.0;
   weight_box[900] := 0.0;
   weight_box[901] := 0.0;
   weight_box[902] := 0.0;
   weight_box[903] := 0.0;
   weight_box[904] := 0.0;
   weight_box[905] := 0.0;
   weight_box[906] := 0.0;
   weight_box[907] := 0.0;
   weight_box[908] := 0.0;
   weight_box[909] := 0.0;
   weight_box[910] := 0.0;
   weight_box[911] := 0.0;
   weight_box[912] := 0.0;
   weight_box[913] := 0.0;
   weight_box[914] := 0.0;
   weight_box[915] := 0.0;
   weight_box[916] := 0.0;
   weight_box[917] := 0.0;
   weight_box[918] := 0.0;
   weight_box[919] := 0.0;
   weight_box[920] := 0.0;
   weight_box[921] := 0.0;
   weight_box[922] := 0.0;
   weight_box[923] := 0.0;
   weight_box[924] := 0.0;
   weight_box[925] := 0.0;
   weight_box[926] := 0.0;
   weight_box[927] := 0.0;
   weight_box[928] := 0.0;
   weight_box[929] := 0.0;
   weight_box[930] := 0.0;
   weight_box[931] := 0.0;
   weight_box[932] := 0.0;
   weight_box[933] := 0.0;
   weight_box[934] := 0.0;
   weight_box[935] := 0.0;
   weight_box[936] := 0.0;
   weight_box[937] := 0.0;
   weight_box[938] := 0.0;
   weight_box[939] := 0.0;
   weight_box[940] := 0.0;
   weight_box[941] := 0.0;
   weight_box[942] := 0.0;
   weight_box[943] := 0.0;
   weight_box[944] := 0.0;
   weight_box[945] := 0.0;
   weight_box[946] := 0.0;
   weight_box[947] := 0.0;
   weight_box[948] := 0.0;
   weight_box[949] := 0.0;
   weight_box[950] := 0.0;
   weight_box[951] := 0.0;
   weight_box[952] := 0.0;
   weight_box[953] := 0.0;
   weight_box[954] := 0.0;
   weight_box[955] := 0.0;
   weight_box[956] := 0.0;
   weight_box[957] := 0.0;
   weight_box[958] := 0.0;
   weight_box[959] := 0.0;
   weight_box[960] := 0.0;
   weight_box[961] := 0.0;
   weight_box[962] := 0.0;
   weight_box[963] := 0.0;
   weight_box[964] := 0.0;
   weight_box[965] := 0.0;
   weight_box[966] := 0.0;
   weight_box[967] := 0.0;
   weight_box[968] := 0.0;
   weight_box[969] := 0.0;
   weight_box[970] := 0.0;
   weight_box[971] := 0.0;
   weight_box[972] := 0.0;
   weight_box[973] := 0.0;
   weight_box[974] := 0.0;
   weight_box[975] := 0.0;
   weight_box[976] := 0.0;
   weight_box[977] := 0.0;
   weight_box[978] := 0.0;
   weight_box[979] := 0.0;
   weight_box[980] := 0.0;
   weight_box[981] := 0.0;
   weight_box[982] := 0.0;
   weight_box[983] := 0.0;
   weight_box[984] := 0.0;
   weight_box[985] := 0.0;
   weight_box[986] := 0.0;
   weight_box[987] := 0.0;
   weight_box[988] := 0.0;
   weight_box[989] := 0.0;
   weight_box[990] := 0.0;
   weight_box[991] := 0.0;
   weight_box[992] := 0.0;
   weight_box[993] := 0.0;
   weight_box[994] := 0.0;
   weight_box[995] := 0.0;
   weight_box[996] := 0.0;
   weight_box[997] := 0.0;
   weight_box[998] := 0.0;
   weight_box[999] := 0.0;
   weight_box[1000] := 0.0;
   weight_box[1001] := 0.0;
   weight_box[1002] := 0.0;
   weight_box[1003] := 0.0;
   weight_box[1004] := 0.0;
   weight_box[1005] := 0.0;
   weight_box[1006] := 0.0;
   weight_box[1007] := 0.0;
   weight_box[1008] := 0.0;
   weight_box[1009] := 0.0;
   weight_box[1010] := 0.0;
   weight_box[1011] := 0.0;
   weight_box[1012] := 0.0;
   weight_box[1013] := 0.0;
   weight_box[1014] := 0.0;
   weight_box[1015] := 0.0;
   weight_box[1016] := 0.0;
   weight_box[1017] := 0.0;
   weight_box[1018] := 0.0;
   weight_box[1019] := 0.0;
   weight_box[1020] := 0.0;
   weight_box[1021] := 0.0;
   weight_box[1022] := 0.0;
   weight_box[1023] := 0.0;
   weight_box[1024] := 0.0;
   weight_box[1025] := 0.0;
   weight_box[1026] := 0.0;
   weight_box[1027] := 0.0;
   weight_box[1028] := 0.0;
   weight_box[1029] := 0.0;
   weight_box[1030] := 0.0;
   weight_box[1031] := 0.0;
   weight_box[1032] := 0.0;
   weight_box[1033] := 0.0;
   weight_box[1034] := 0.0;
   weight_box[1035] := 0.0;
   weight_box[1036] := 0.0;
   weight_box[1037] := 0.0;
   weight_box[1038] := 0.0;
   weight_box[1039] := 0.0;
   weight_box[1040] := 0.0;
   weight_box[1041] := 0.0;
   weight_box[1042] := 0.0;
   weight_box[1043] := 0.0;
   weight_box[1044] := 0.0;
   weight_box[1045] := 0.0;
   weight_box[1046] := 0.0;
   weight_box[1047] := 0.0;
   weight_box[1048] := 0.0;
   weight_box[1049] := 0.0;
   weight_box[1050] := 0.0;
   weight_box[1051] := 0.0;
   weight_box[1052] := 0.0;
   weight_box[1053] := 0.0;
   weight_box[1054] := 0.0;
   weight_box[1055] := 0.0;
   weight_box[1056] := 0.0;
   weight_box[1057] := 0.0;
   weight_box[1058] := 0.0;
   weight_box[1059] := 0.0;
   weight_box[1060] := 0.0;
   weight_box[1061] := 0.0;
   weight_box[1062] := 0.0;
   weight_box[1063] := 0.0;
   weight_box[1064] := 0.0;
   weight_box[1065] := 0.0;
   weight_box[1066] := 0.0;
   weight_box[1067] := 0.0;
   weight_box[1068] := 0.0;
   weight_box[1069] := 0.0;
   weight_box[1070] := 0.0;
   weight_box[1071] := 0.0;
   weight_box[1072] := 0.0;
   weight_box[1073] := 0.0;
   weight_box[1074] := 0.0;
   weight_box[1075] := 0.0;
   weight_box[1076] := 0.0;
   weight_box[1077] := 0.0;
   weight_box[1078] := 0.0;
   weight_box[1079] := 0.0;
   weight_box[1080] := 0.0;
   weight_box[1081] := 0.0;
   weight_box[1082] := 0.0;
   weight_box[1083] := 0.0;
   weight_box[1084] := 0.0;
   weight_box[1085] := 0.0;
   weight_box[1086] := 0.0;
   weight_box[1087] := 0.0;
   weight_box[1088] := 0.0;
   weight_box[1089] := 0.0;
   weight_box[1090] := 0.0;
   weight_box[1091] := 0.0;
   weight_box[1092] := 0.0;
   weight_box[1093] := 0.0;
   weight_box[1094] := 0.0;
   weight_box[1095] := 0.0;
   weight_box[1096] := 0.0;
   weight_box[1097] := 0.0;
   weight_box[1098] := 0.0;
   weight_box[1099] := 0.0;
   weight_box[1100] := 0.0;
   weight_box[1101] := 0.0;
   weight_box[1102] := 0.0;
   weight_box[1103] := 0.0;
   weight_box[1104] := 0.0;
   weight_box[1105] := 0.0;
   weight_box[1106] := 0.0;
   weight_box[1107] := 0.0;
   weight_box[1108] := 0.0;
   weight_box[1109] := 0.0;
   weight_box[1110] := 0.0;
   weight_box[1111] := 0.0;
   weight_box[1112] := 0.0;
   weight_box[1113] := 0.0;
   weight_box[1114] := 0.0;
   weight_box[1115] := 0.0;
   weight_box[1116] := 0.0;
   weight_box[1117] := 0.0;
   weight_box[1118] := 0.0;
   weight_box[1119] := 0.0;
   weight_box[1120] := 0.0;
   weight_box[1121] := 0.0;
   weight_box[1122] := 0.0;
   weight_box[1123] := 0.0;
   weight_box[1124] := 0.0;
   weight_box[1125] := 0.0;
   weight_box[1126] := 0.0;
   weight_box[1127] := 0.0;
   weight_box[1128] := 0.0;
   weight_box[1129] := 0.0;
   weight_box[1130] := 0.0;
   weight_box[1131] := 0.0;
   weight_box[1132] := 0.0;
   weight_box[1133] := 0.0;
   weight_box[1134] := 0.0;
   weight_box[1135] := 0.0;
   weight_box[1136] := 0.0;
   weight_box[1137] := 0.0;
   weight_box[1138] := 0.0;
   weight_box[1139] := 0.0;
   weight_box[1140] := 0.0;
   weight_box[1141] := 0.0;
   weight_box[1142] := 0.0;
   weight_box[1143] := 0.0;
   weight_box[1144] := 0.0;
   weight_box[1145] := 0.0;
   weight_box[1146] := 0.0;
   weight_box[1147] := 0.0;
   weight_box[1148] := 0.0;
   weight_box[1149] := 0.0;
   weight_box[1150] := 0.0;
   weight_box[1151] := 0.0;
   weight_box[1152] := 0.0;
   weight_box[1153] := 0.0;
   weight_box[1154] := 0.0;
   weight_box[1155] := 0.0;
   weight_box[1156] := 0.0;
   weight_box[1157] := 0.0;
   weight_box[1158] := 0.0;
   weight_box[1159] := 0.0;
   weight_box[1160] := 0.0;
   weight_box[1161] := 0.0;
   weight_box[1162] := 0.0;
   weight_box[1163] := 0.0;
   weight_box[1164] := 0.0;
   weight_box[1165] := 0.0;
   weight_box[1166] := 0.0;
   weight_box[1167] := 0.0;
   weight_box[1168] := 0.0;
   weight_box[1169] := 0.0;
   weight_box[1170] := 0.0;
   weight_box[1171] := 0.0;
   weight_box[1172] := 0.0;
   weight_box[1173] := 0.0;
   weight_box[1174] := 0.0;
   weight_box[1175] := 0.0;
   weight_box[1176] := 0.0;
   weight_box[1177] := 0.0;
   weight_box[1178] := 0.0;
   weight_box[1179] := 0.0;
   weight_box[1180] := 0.0;
   weight_box[1181] := 0.0;
   weight_box[1182] := 0.0;
   weight_box[1183] := 0.0;
   weight_box[1184] := 0.0;
   weight_box[1185] := 0.0;
   weight_box[1186] := 0.0;
   weight_box[1187] := 0.0;
   weight_box[1188] := 0.0;
   weight_box[1189] := 0.0;
   weight_box[1190] := 0.0;
   weight_box[1191] := 0.0;
   weight_box[1192] := 0.0;
   weight_box[1193] := 0.0;
   weight_box[1194] := 0.0;
   weight_box[1195] := 0.0;
   weight_box[1196] := 0.0;
   weight_box[1197] := 0.0;
   weight_box[1198] := 0.0;
   weight_box[1199] := 0.0;
   weight_box[1200] := 0.0;
   weight_box[1201] := 0.0;
   weight_box[1202] := 0.0;
   weight_box[1203] := 0.0;
   weight_box[1204] := 0.0;
   weight_box[1205] := 0.0;
   weight_box[1206] := 0.0;
   weight_box[1207] := 0.0;
   weight_box[1208] := 0.0;
   weight_box[1209] := 0.0;
   weight_box[1210] := 0.0;
   weight_box[1211] := 0.0;
   weight_box[1212] := 0.0;
   weight_box[1213] := 0.0;
   weight_box[1214] := 0.0;
   weight_box[1215] := 0.0;
   weight_box[1216] := 0.0;
   weight_box[1217] := 0.0;
   weight_box[1218] := 0.0;
   weight_box[1219] := 0.0;
   weight_box[1220] := 0.0;
   weight_box[1221] := 0.0;
   weight_box[1222] := 0.0;
   weight_box[1223] := 0.0;
   weight_box[1224] := 0.0;
   weight_box[1225] := 0.0;
   weight_box[1226] := 0.0;
   weight_box[1227] := 0.0;
   weight_box[1228] := 0.0;
   weight_box[1229] := 0.0;
   weight_box[1230] := 0.0;
   weight_box[1231] := 0.0;
   weight_box[1232] := 0.0;
   weight_box[1233] := 0.0;
   weight_box[1234] := 0.0;
   weight_box[1235] := 0.0;
   weight_box[1236] := 0.0;
   weight_box[1237] := 0.0;
   weight_box[1238] := 0.0;
   weight_box[1239] := 0.0;
   weight_box[1240] := 0.0;
   weight_box[1241] := 0.0;
   weight_box[1242] := 0.0;
   weight_box[1243] := 0.0;
   weight_box[1244] := 0.0;
   weight_box[1245] := 0.0;
   weight_box[1246] := 0.0;
   weight_box[1247] := 0.0;
   weight_box[1248] := 0.0;
   weight_box[1249] := 0.0;
   weight_box[1250] := 0.0;
   weight_box[1251] := 0.0;
   weight_box[1252] := 0.0;
   weight_box[1253] := 0.0;
   weight_box[1254] := 0.0;
   weight_box[1255] := 0.0;
   weight_box[1256] := 0.0;
   weight_box[1257] := 0.0;
   weight_box[1258] := 0.0;
   weight_box[1259] := 0.0;
   weight_box[1260] := 0.0;
   weight_box[1261] := 0.0;
   weight_box[1262] := 0.0;
   weight_box[1263] := 0.0;
   weight_box[1264] := 0.0;
   weight_box[1265] := 0.0;
   weight_box[1266] := 0.0;
   weight_box[1267] := 0.0;
   weight_box[1268] := 0.0;
   weight_box[1269] := 0.0;
   weight_box[1270] := 0.0;
   weight_box[1271] := 0.0;
   weight_box[1272] := 0.0;
   weight_box[1273] := 0.0;
   weight_box[1274] := 0.0;
   weight_box[1275] := 0.0;
   weight_box[1276] := 0.0;
   weight_box[1277] := 0.0;
   weight_box[1278] := 0.0;
   weight_box[1279] := 0.0;
   weight_box[1280] := 0.0;
   weight_box[1281] := 0.0;
   weight_box[1282] := 0.0;
   weight_box[1283] := 0.0;
   weight_box[1284] := 0.0;
   weight_box[1285] := 0.0;
   weight_box[1286] := 0.0;
   weight_box[1287] := 0.0;
   weight_box[1288] := 0.0;
   weight_box[1289] := 0.0;
   weight_box[1290] := 0.0;
   weight_box[1291] := 0.0;
   weight_box[1292] := 0.0;
   weight_box[1293] := 0.0;
   weight_box[1294] := 0.0;
   weight_box[1295] := 0.0;
   weight_box[1296] := 0.0;
   weight_box[1297] := 0.0;
   weight_box[1298] := 0.0;
   weight_box[1299] := 0.0;
   weight_box[1300] := 0.0;
   weight_box[1301] := 0.0;
   weight_box[1302] := 0.0;
   weight_box[1303] := 0.0;
   weight_box[1304] := 0.0;
   weight_box[1305] := 0.0;
   weight_box[1306] := 0.0;
   weight_box[1307] := 0.0;
   weight_box[1308] := 0.0;
   weight_box[1309] := 0.0;
   weight_box[1310] := 0.0;
   weight_box[1311] := 0.0;
   weight_box[1312] := 0.0;
   weight_box[1313] := 0.0;
   weight_box[1314] := 0.0;
   weight_box[1315] := 0.0;
   weight_box[1316] := 0.0;
   weight_box[1317] := 0.0;
   weight_box[1318] := 0.0;
   weight_box[1319] := 0.0;
   weight_box[1320] := 0.0;
   weight_box[1321] := 0.0;
   weight_box[1322] := 0.0;
   weight_box[1323] := 0.0;
   weight_box[1324] := 0.0;
   weight_box[1325] := 0.0;
   weight_box[1326] := 0.0;
   weight_box[1327] := 0.0;
   weight_box[1328] := 0.0;
   weight_box[1329] := 0.0;
   weight_box[1330] := 0.0;
   weight_box[1331] := 0.0;
   weight_box[1332] := 0.0;
   weight_box[1333] := 0.0;
   weight_box[1334] := 0.0;
   weight_box[1335] := 0.0;
   weight_box[1336] := 0.0;
   weight_box[1337] := 0.0;
   weight_box[1338] := 0.0;
   weight_box[1339] := 0.0;
   weight_box[1340] := 0.0;
   weight_box[1341] := 0.0;
   weight_box[1342] := 0.0;
   weight_box[1343] := 0.0;
   weight_box[1344] := 0.0;
   weight_box[1345] := 0.0;
   weight_box[1346] := 0.0;
   weight_box[1347] := 0.0;
   weight_box[1348] := 0.0;
   weight_box[1349] := 0.0;
   weight_box[1350] := 0.0;
   weight_box[1351] := 0.0;
   weight_box[1352] := 0.0;
   weight_box[1353] := 0.0;
   weight_box[1354] := 0.0;
   weight_box[1355] := 0.0;
   weight_box[1356] := 0.0;
   weight_box[1357] := 0.0;
   weight_box[1358] := 0.0;
   weight_box[1359] := 0.0;
   weight_box[1360] := 0.0;
   weight_box[1361] := 0.0;
   weight_box[1362] := 0.0;
   weight_box[1363] := 0.0;
   weight_box[1364] := 0.0;
   weight_box[1365] := 0.0;
   weight_box[1366] := 0.0;
   weight_box[1367] := 0.0;
   weight_box[1368] := 0.0;
   weight_box[1369] := 0.0;
   weight_box[1370] := 0.0;
   weight_box[1371] := 0.0;
   weight_box[1372] := 0.0;
   weight_box[1373] := 0.0;
   weight_box[1374] := 0.0;
   weight_box[1375] := 0.0;
   weight_box[1376] := 0.0;
   weight_box[1377] := 0.0;
   weight_box[1378] := 0.0;
   weight_box[1379] := 0.0;
   weight_box[1380] := 0.0;
   weight_box[1381] := 0.0;
   weight_box[1382] := 0.0;
   weight_box[1383] := 0.0;
   weight_box[1384] := 0.0;
   weight_box[1385] := 0.0;
   weight_box[1386] := 0.0;
   weight_box[1387] := 0.0;
   weight_box[1388] := 0.0;
   weight_box[1389] := 0.0;
   weight_box[1390] := 0.0;
   weight_box[1391] := 0.0;
   weight_box[1392] := 0.0;
   weight_box[1393] := 0.0;
   weight_box[1394] := 0.0;
   weight_box[1395] := 0.0;
   weight_box[1396] := 0.0;
   weight_box[1397] := 0.0;
   weight_box[1398] := 0.0;
   weight_box[1399] := 0.0;
   weight_box[1400] := 0.0;
   weight_box[1401] := 0.0;
   weight_box[1402] := 0.0;
   weight_box[1403] := 0.0;
   weight_box[1404] := 0.0;
   weight_box[1405] := 0.0;
   weight_box[1406] := 0.0;
   weight_box[1407] := 0.0;
   weight_box[1408] := 0.0;
   weight_box[1409] := 0.0;
   weight_box[1410] := 0.0;
   weight_box[1411] := 0.0;
   weight_box[1412] := 0.0;
   weight_box[1413] := 0.0;
   weight_box[1414] := 0.0;
   weight_box[1415] := 0.0;
   weight_box[1416] := 0.0;
   weight_box[1417] := 0.0;
   weight_box[1418] := 0.0;
   weight_box[1419] := 0.0;
   weight_box[1420] := 0.0;
   weight_box[1421] := 0.0;
   weight_box[1422] := 0.0;
   weight_box[1423] := 0.0;
   weight_box[1424] := 0.0;
   weight_box[1425] := 0.0;
   weight_box[1426] := 0.0;
   weight_box[1427] := 0.0;
   weight_box[1428] := 0.0;
   weight_box[1429] := 0.0;
   weight_box[1430] := 0.0;
   weight_box[1431] := 0.0;
   weight_box[1432] := 0.0;
   weight_box[1433] := 0.0;
   weight_box[1434] := 0.0;
   weight_box[1435] := 0.0;
   weight_box[1436] := 0.0;
   weight_box[1437] := 0.0;
   weight_box[1438] := 0.0;
   weight_box[1439] := 0.0;
   weight_box[1440] := 0.0;
   weight_box[1441] := 0.0;
   weight_box[1442] := 0.0;
   weight_box[1443] := 0.0;
   weight_box[1444] := 0.0;
   weight_box[1445] := 0.0;
   weight_box[1446] := 0.0;
   weight_box[1447] := 0.0;
   weight_box[1448] := 0.0;
   weight_box[1449] := 0.0;
   weight_box[1450] := 0.0;
   weight_box[1451] := 0.0;
   weight_box[1452] := 0.0;
   weight_box[1453] := 0.0;
   weight_box[1454] := 0.0;
   weight_box[1455] := 0.0;
   weight_box[1456] := 0.0;
   weight_box[1457] := 0.0;
   weight_box[1458] := 0.0;
   weight_box[1459] := 0.0;
   weight_box[1460] := 0.0;
   weight_box[1461] := 0.0;
   weight_box[1462] := 0.0;
   weight_box[1463] := 0.0;
   weight_box[1464] := 0.0;
   weight_box[1465] := 0.0;
   weight_box[1466] := 0.0;
   weight_box[1467] := 0.0;
   weight_box[1468] := 0.0;
   weight_box[1469] := 0.0;
   weight_box[1470] := 0.0;
   weight_box[1471] := 0.0;
   weight_box[1472] := 0.0;
   weight_box[1473] := 0.0;
   weight_box[1474] := 0.0;
   weight_box[1475] := 0.0;
   weight_box[1476] := 0.0;
   weight_box[1477] := 0.0;
   weight_box[1478] := 0.0;
   weight_box[1479] := 0.0;
   weight_box[1480] := 0.0;
   weight_box[1481] := 0.0;
   weight_box[1482] := 0.0;
   weight_box[1483] := 0.0;
   weight_box[1484] := 0.0;
   weight_box[1485] := 0.0;
   weight_box[1486] := 0.0;
   weight_box[1487] := 0.0;
   weight_box[1488] := 0.0;
   weight_box[1489] := 0.0;
   weight_box[1490] := 0.0;
   weight_box[1491] := 0.0;
   weight_box[1492] := 0.0;
   weight_box[1493] := 0.0;
   weight_box[1494] := 0.0;
   weight_box[1495] := 0.0;
   weight_box[1496] := 0.0;
   weight_box[1497] := 0.0;
   weight_box[1498] := 0.0;
   weight_box[1499] := 0.0;
   weight_box[1500] := 0.0;
   weight_box[1501] := 0.0;
   weight_box[1502] := 0.0;
   weight_box[1503] := 0.0;
   weight_box[1504] := 0.0;
   weight_box[1505] := 0.0;
   weight_box[1506] := 0.0;
   weight_box[1507] := 0.0;
   weight_box[1508] := 0.0;
   weight_box[1509] := 0.0;
   weight_box[1510] := 0.0;
   weight_box[1511] := 0.0;
   weight_box[1512] := 0.0;
   weight_box[1513] := 0.0;
   weight_box[1514] := 0.0;
   weight_box[1515] := 0.0;
   weight_box[1516] := 0.0;
   weight_box[1517] := 0.0;
   weight_box[1518] := 0.0;
   weight_box[1519] := 0.0;
   weight_box[1520] := 0.0;
   weight_box[1521] := 0.0;
   weight_box[1522] := 0.0;
   weight_box[1523] := 0.0;
   weight_box[1524] := 0.0;
   weight_box[1525] := 0.0;
   weight_box[1526] := 0.0;
   weight_box[1527] := 0.0;
   weight_box[1528] := 0.0;
   weight_box[1529] := 0.0;
   weight_box[1530] := 0.0;
   weight_box[1531] := 0.0;
   weight_box[1532] := 0.0;
   weight_box[1533] := 0.0;
   weight_box[1534] := 0.0;
   weight_box[1535] := 0.0;
   weight_box[1536] := 0.0;
   weight_box[1537] := 0.0;
   weight_box[1538] := 0.0;
   weight_box[1539] := 0.0;
   weight_box[1540] := 0.0;
   weight_box[1541] := 0.0;
   weight_box[1542] := 0.0;
   weight_box[1543] := 0.0;
   weight_box[1544] := 0.0;
   weight_box[1545] := 0.0;
   weight_box[1546] := 0.0;
   weight_box[1547] := 0.0;
   weight_box[1548] := 0.0;
   weight_box[1549] := 0.0;
   weight_box[1550] := 0.0;
   weight_box[1551] := 0.0;
   weight_box[1552] := 0.0;
   weight_box[1553] := 0.0;
   weight_box[1554] := 0.0;
   weight_box[1555] := 0.0;
   weight_box[1556] := 0.0;
   weight_box[1557] := 0.0;
   weight_box[1558] := 0.0;
   weight_box[1559] := 0.0;
   weight_box[1560] := 0.0;
   weight_box[1561] := 0.0;
   weight_box[1562] := 0.0;
   weight_box[1563] := 0.0;
   weight_box[1564] := 0.0;
   weight_box[1565] := 0.0;
   weight_box[1566] := 0.0;
   weight_box[1567] := 0.0;
   weight_box[1568] := 0.0;
   weight_box[1569] := 0.0;
   weight_box[1570] := 0.0;
   weight_box[1571] := 0.0;
   weight_box[1572] := 0.0;
   weight_box[1573] := 0.0;
   weight_box[1574] := 0.0;
   weight_box[1575] := 0.0;
   weight_box[1576] := 0.0;
   weight_box[1577] := 0.0;
   weight_box[1578] := 0.0;
   weight_box[1579] := 0.0;
   weight_box[1580] := 0.0;
   weight_box[1581] := 0.0;
   weight_box[1582] := 0.0;
   weight_box[1583] := 0.0;
   weight_box[1584] := 0.0;
   weight_box[1585] := 0.0;
   weight_box[1586] := 0.0;
   weight_box[1587] := 0.0;
   weight_box[1588] := 0.0;
   weight_box[1589] := 0.0;
   weight_box[1590] := 0.0;
   weight_box[1591] := 0.0;
   weight_box[1592] := 0.0;
   weight_box[1593] := 0.0;
   weight_box[1594] := 0.0;
   weight_box[1595] := 0.0;
   weight_box[1596] := 0.0;
   weight_box[1597] := 0.0;
   weight_box[1598] := 0.0;
   weight_box[1599] := 0.0;
   weight_box[1600] := 0.0;
   weight_box[1601] := 0.0;
   weight_box[1602] := 0.0;
   weight_box[1603] := 0.0;
   weight_box[1604] := 0.0;
   weight_box[1605] := 0.0;
   weight_box[1606] := 0.0;
   weight_box[1607] := 0.0;
   weight_box[1608] := 0.0;
   weight_box[1609] := 0.0;
   weight_box[1610] := 0.0;
   weight_box[1611] := 0.0;
   weight_box[1612] := 0.0;
   weight_box[1613] := 0.0;
   weight_box[1614] := 0.0;
   weight_box[1615] := 0.0;
   weight_box[1616] := 0.0;
   weight_box[1617] := 0.0;
   weight_box[1618] := 0.0;
   weight_box[1619] := 0.0;
   weight_box[1620] := 0.0;
   weight_box[1621] := 0.0;
   weight_box[1622] := 0.0;
   weight_box[1623] := 0.0;
   weight_box[1624] := 0.0;
   weight_box[1625] := 0.0;
   weight_box[1626] := 0.0;
   weight_box[1627] := 0.0;
   weight_box[1628] := 0.0;
   weight_box[1629] := 0.0;
   weight_box[1630] := 0.0;
   weight_box[1631] := 0.0;
   weight_box[1632] := 0.0;
   weight_box[1633] := 0.0;
   weight_box[1634] := 0.0;
   weight_box[1635] := 0.0;
   weight_box[1636] := 0.0;
   weight_box[1637] := 0.0;
   weight_box[1638] := 0.0;
   weight_box[1639] := 0.0;
   weight_box[1640] := 0.0;
   weight_box[1641] := 0.0;
   weight_box[1642] := 0.0;
   weight_box[1643] := 0.0;
   weight_box[1644] := 0.0;
   weight_box[1645] := 0.0;
   weight_box[1646] := 0.0;
   weight_box[1647] := 0.0;
   weight_box[1648] := 0.0;
   weight_box[1649] := 0.0;
   weight_box[1650] := 0.0;
   weight_box[1651] := 0.0;
   weight_box[1652] := 0.0;
   weight_box[1653] := 0.0;
   weight_box[1654] := 0.0;
   weight_box[1655] := 0.0;
   weight_box[1656] := 0.0;
   weight_box[1657] := 0.0;
   weight_box[1658] := 0.0;
   weight_box[1659] := 0.0;
   weight_box[1660] := 0.0;
   weight_box[1661] := 0.0;
   weight_box[1662] := 0.0;
   weight_box[1663] := 0.0;
   weight_box[1664] := 0.0;
   weight_box[1665] := 0.0;
   weight_box[1666] := 0.0;
   weight_box[1667] := 0.0;
   weight_box[1668] := 0.0;
   weight_box[1669] := 0.0;
   weight_box[1670] := 0.0;
   weight_box[1671] := 0.0;
   weight_box[1672] := 0.0;
   weight_box[1673] := 0.0;
   weight_box[1674] := 0.0;
   weight_box[1675] := 0.0;
   weight_box[1676] := 0.0;
   weight_box[1677] := 0.0;
   weight_box[1678] := 0.0;
   weight_box[1679] := 0.0;
   weight_box[1680] := 0.0;
   weight_box[1681] := 0.0;
   weight_box[1682] := 0.0;
   weight_box[1683] := 0.0;
   weight_box[1684] := 0.0;
   weight_box[1685] := 0.0;
   weight_box[1686] := 0.0;
   weight_box[1687] := 0.0;
   weight_box[1688] := 0.0;
   weight_box[1689] := 0.0;
   weight_box[1690] := 0.0;
   weight_box[1691] := 0.0;
   weight_box[1692] := 0.0;
   weight_box[1693] := 0.0;
   weight_box[1694] := 0.0;
   weight_box[1695] := 0.0;
   weight_box[1696] := 0.0;
   weight_box[1697] := 0.0;
   weight_box[1698] := 0.0;
   weight_box[1699] := 0.0;
   weight_box[1700] := 0.0;
   weight_box[1701] := 0.0;
   weight_box[1702] := 0.0;
   weight_box[1703] := 0.0;
   weight_box[1704] := 0.0;
   weight_box[1705] := 0.0;
   weight_box[1706] := 0.0;
   weight_box[1707] := 0.0;
   weight_box[1708] := 0.0;
   weight_box[1709] := 0.0;
   weight_box[1710] := 0.0;
   weight_box[1711] := 0.0;
   weight_box[1712] := 0.0;
   weight_box[1713] := 0.0;
   weight_box[1714] := 0.0;
   weight_box[1715] := 0.0;
   weight_box[1716] := 0.0;
   weight_box[1717] := 0.0;
   weight_box[1718] := 0.0;
   weight_box[1719] := 0.0;
   weight_box[1720] := 0.0;
   weight_box[1721] := 0.0;
   weight_box[1722] := 0.0;
   weight_box[1723] := 0.0;
   weight_box[1724] := 0.0;
   weight_box[1725] := 0.0;
   weight_box[1726] := 0.0;
   weight_box[1727] := 0.0;
   weight_box[1728] := 0.0;
   weight_box[1729] := 0.0;
   weight_box[1730] := 0.0;
   weight_box[1731] := 0.0;
   weight_box[1732] := 0.0;
   weight_box[1733] := 0.0;
   weight_box[1734] := 0.0;
   weight_box[1735] := 0.0;
   weight_box[1736] := 0.0;
   weight_box[1737] := 0.0;
   weight_box[1738] := 0.0;
   weight_box[1739] := 0.0;
   weight_box[1740] := 0.0;
   weight_box[1741] := 0.0;
   weight_box[1742] := 0.0;
   weight_box[1743] := 0.0;
   weight_box[1744] := 0.0;
   weight_box[1745] := 0.0;
   weight_box[1746] := 0.0;
   weight_box[1747] := 0.0;
   weight_box[1748] := 0.0;
   weight_box[1749] := 0.0;
   weight_box[1750] := 0.0;
   weight_box[1751] := 0.0;
   weight_box[1752] := 0.0;
   weight_box[1753] := 0.0;
   weight_box[1754] := 0.0;
   weight_box[1755] := 0.0;
   weight_box[1756] := 0.0;
   weight_box[1757] := 0.0;
   weight_box[1758] := 0.0;
   weight_box[1759] := 0.0;
   weight_box[1760] := 0.0;
   weight_box[1761] := 0.0;
   weight_box[1762] := 0.0;
   weight_box[1763] := 0.0;
   weight_box[1764] := 0.0;
   weight_box[1765] := 0.0;
   weight_box[1766] := 0.0;
   weight_box[1767] := 0.0;
   weight_box[1768] := 0.0;
   weight_box[1769] := 0.0;
   weight_box[1770] := 0.0;
   weight_box[1771] := 0.0;
   weight_box[1772] := 0.0;
   weight_box[1773] := 0.0;
   weight_box[1774] := 0.0;
   weight_box[1775] := 0.0;
   weight_box[1776] := 0.0;
   weight_box[1777] := 0.0;
   weight_box[1778] := 0.0;
   weight_box[1779] := 0.0;
   weight_box[1780] := 0.0;
   weight_box[1781] := 0.0;
   weight_box[1782] := 0.0;
   weight_box[1783] := 0.0;
   weight_box[1784] := 0.0;
   weight_box[1785] := 0.0;
   weight_box[1786] := 0.0;
   weight_box[1787] := 0.0;
   weight_box[1788] := 0.0;
   weight_box[1789] := 0.0;
   weight_box[1790] := 0.0;
   weight_box[1791] := 0.0;
   weight_box[1792] := 0.0;
   weight_box[1793] := 0.0;
   weight_box[1794] := 0.0;
   weight_box[1795] := 0.0;
   weight_box[1796] := 0.0;
   weight_box[1797] := 0.0;
   weight_box[1798] := 0.0;
   weight_box[1799] := 0.0;
   weight_box[1800] := 0.0;
   weight_box[1801] := 0.0;
   weight_box[1802] := 0.0;
   weight_box[1803] := 0.0;
   weight_box[1804] := 0.0;
   weight_box[1805] := 0.0;
   weight_box[1806] := 0.0;
   weight_box[1807] := 0.0;
   weight_box[1808] := 0.0;
   weight_box[1809] := 0.0;
   weight_box[1810] := 0.0;
   weight_box[1811] := 0.0;
   weight_box[1812] := 0.0;
   weight_box[1813] := 0.0;
   weight_box[1814] := 0.0;
   weight_box[1815] := 0.0;
   weight_box[1816] := 0.0;
   weight_box[1817] := 0.0;
   weight_box[1818] := 0.0;
   weight_box[1819] := 0.0;
   weight_box[1820] := 0.0;
   weight_box[1821] := 0.0;
   weight_box[1822] := 0.0;
   weight_box[1823] := 0.0;
   weight_box[1824] := 0.0;
   weight_box[1825] := 0.0;
   weight_box[1826] := 0.0;
   weight_box[1827] := 0.0;
   weight_box[1828] := 0.0;
   weight_box[1829] := 0.0;
   weight_box[1830] := 0.0;
   weight_box[1831] := 0.0;
   weight_box[1832] := 0.0;
   weight_box[1833] := 0.0;
   weight_box[1834] := 0.0;
   weight_box[1835] := 0.0;
   weight_box[1836] := 0.0;
   weight_box[1837] := 0.0;
   weight_box[1838] := 0.0;
   weight_box[1839] := 0.0;
   weight_box[1840] := 0.0;
   weight_box[1841] := 0.0;
   weight_box[1842] := 0.0;
   weight_box[1843] := 0.0;
   weight_box[1844] := 0.0;
   weight_box[1845] := 0.0;
   weight_box[1846] := 0.0;
   weight_box[1847] := 0.0;
   weight_box[1848] := 0.0;
   weight_box[1849] := 0.0;
   weight_box[1850] := 0.0;
   weight_box[1851] := 0.0;
   weight_box[1852] := 0.0;
   weight_box[1853] := 0.0;
   weight_box[1854] := 0.0;
   weight_box[1855] := 0.0;
   weight_box[1856] := 0.0;
   weight_box[1857] := 0.0;
   weight_box[1858] := 0.0;
   weight_box[1859] := 0.0;
   weight_box[1860] := 0.0;
   weight_box[1861] := 0.0;
   weight_box[1862] := 0.0;
   weight_box[1863] := 0.0;
   weight_box[1864] := 0.0;
   weight_box[1865] := 0.0;
   weight_box[1866] := 0.0;
   weight_box[1867] := 0.0;
   weight_box[1868] := 0.0;
   weight_box[1869] := 0.0;
   weight_box[1870] := 0.0;
   weight_box[1871] := 0.0;
   weight_box[1872] := 0.0;
   weight_box[1873] := 0.0;
   weight_box[1874] := 0.0;
   weight_box[1875] := 0.0;
   weight_box[1876] := 0.0;
   weight_box[1877] := 0.0;
   weight_box[1878] := 0.0;
   weight_box[1879] := 0.0;
   weight_box[1880] := 0.0;
   weight_box[1881] := 0.0;
   weight_box[1882] := 0.0;
   weight_box[1883] := 0.0;
   weight_box[1884] := 0.0;
   weight_box[1885] := 0.0;
   weight_box[1886] := 0.0;
   weight_box[1887] := 0.0;
   weight_box[1888] := 0.0;
   weight_box[1889] := 0.0;
   weight_box[1890] := 0.0;
   weight_box[1891] := 0.0;
   weight_box[1892] := 0.0;
   weight_box[1893] := 0.0;
   weight_box[1894] := 0.0;
   weight_box[1895] := 0.0;
   weight_box[1896] := 0.0;
   weight_box[1897] := 0.0;
   weight_box[1898] := 0.0;
   weight_box[1899] := 0.0;
   weight_box[1900] := 0.0;
   weight_box[1901] := 0.0;
   weight_box[1902] := 0.0;
   weight_box[1903] := 0.0;
   weight_box[1904] := 0.0;
   weight_box[1905] := 0.0;
   weight_box[1906] := 0.0;
   weight_box[1907] := 0.0;
   weight_box[1908] := 0.0;
   weight_box[1909] := 0.0;
   weight_box[1910] := 0.0;
   weight_box[1911] := 0.0;
   weight_box[1912] := 0.0;
   weight_box[1913] := 0.0;
   weight_box[1914] := 0.0;
   weight_box[1915] := 0.0;
   weight_box[1916] := 0.0;
   weight_box[1917] := 0.0;
   weight_box[1918] := 0.0;
   weight_box[1919] := 0.0;
   weight_box[1920] := 0.0;
   weight_box[1921] := 0.0;
   weight_box[1922] := 0.0;
   weight_box[1923] := 0.0;
   weight_box[1924] := 0.0;
   weight_box[1925] := 0.0;
   weight_box[1926] := 0.0;
   weight_box[1927] := 0.0;
   weight_box[1928] := 0.0;
   weight_box[1929] := 0.0;
   weight_box[1930] := 0.0;
   weight_box[1931] := 0.0;
   weight_box[1932] := 0.0;
   weight_box[1933] := 0.0;
   weight_box[1934] := 0.0;
   weight_box[1935] := 0.0;
   weight_box[1936] := 0.0;
   weight_box[1937] := 0.0;
   weight_box[1938] := 0.0;
   weight_box[1939] := 0.0;
   weight_box[1940] := 0.0;
   weight_box[1941] := 0.0;
   weight_box[1942] := 0.0;
   weight_box[1943] := 0.0;
   weight_box[1944] := 0.0;
   weight_box[1945] := 0.0;
   weight_box[1946] := 0.0;
   weight_box[1947] := 0.0;
   weight_box[1948] := 0.0;
   weight_box[1949] := 0.0;
   weight_box[1950] := 0.0;
   weight_box[1951] := 0.0;
   weight_box[1952] := 0.0;
   weight_box[1953] := 0.0;
   weight_box[1954] := 0.0;
   weight_box[1955] := 0.0;
   weight_box[1956] := 0.0;
   weight_box[1957] := 0.0;
   weight_box[1958] := 0.0;
   weight_box[1959] := 0.0;
   weight_box[1960] := 0.0;
   weight_box[1961] := 0.0;
   weight_box[1962] := 0.0;
   weight_box[1963] := 0.0;
   weight_box[1964] := 0.0;
   weight_box[1965] := 0.0;
   weight_box[1966] := 0.0;
   weight_box[1967] := 0.0;
   weight_box[1968] := 0.0;
   weight_box[1969] := 0.0;
   weight_box[1970] := 0.0;
   weight_box[1971] := 0.0;
   weight_box[1972] := 0.0;
   weight_box[1973] := 0.0;
   weight_box[1974] := 0.0;
   weight_box[1975] := 0.0;
   weight_box[1976] := 0.0;
   weight_box[1977] := 0.0;
   weight_box[1978] := 0.0;
   weight_box[1979] := 0.0;
   weight_box[1980] := 0.0;
   weight_box[1981] := 0.0;
   weight_box[1982] := 0.0;
   weight_box[1983] := 0.0;
   weight_box[1984] := 0.0;
   weight_box[1985] := 0.0;
   weight_box[1986] := 0.0;
   weight_box[1987] := 0.0;
   weight_box[1988] := 0.0;
   weight_box[1989] := 0.0;
   weight_box[1990] := 0.0;
   weight_box[1991] := 0.0;
   weight_box[1992] := 0.0;
   weight_box[1993] := 0.0;
   weight_box[1994] := 0.0;
   weight_box[1995] := 0.0;
   weight_box[1996] := 0.0;
   weight_box[1997] := 0.0;
   weight_box[1998] := 0.0;
   weight_box[1999] := 0.0;
   weight_box[2000] := 0.0;
   weight_box[2001] := 0.0;
   weight_box[2002] := 0.0;
   weight_box[2003] := 0.0;
   weight_box[2004] := 0.0;
   weight_box[2005] := 0.0;
   weight_box[2006] := 0.0;
   weight_box[2007] := 0.0;
   weight_box[2008] := 0.0;
   weight_box[2009] := 0.0;
   weight_box[2010] := 0.0;
   weight_box[2011] := 0.0;
   weight_box[2012] := 0.0;
   weight_box[2013] := 0.0;
   weight_box[2014] := 0.0;
   weight_box[2015] := 0.0;
   weight_box[2016] := 0.0;
   weight_box[2017] := 0.0;
   weight_box[2018] := 0.0;
   weight_box[2019] := 0.0;
   weight_box[2020] := 0.0;
   weight_box[2021] := 0.0;
   weight_box[2022] := 0.0;
   weight_box[2023] := 0.0;
   weight_box[2024] := 0.0;
   weight_box[2025] := 0.0;
   weight_box[2026] := 0.0;
   weight_box[2027] := 0.0;
   weight_box[2028] := 0.0;
   weight_box[2029] := 0.0;
   weight_box[2030] := 0.0;
   weight_box[2031] := 0.0;
   weight_box[2032] := 0.0;
   weight_box[2033] := 0.0;
   weight_box[2034] := 0.0;
   weight_box[2035] := 0.0;
   weight_box[2036] := 0.0;
   weight_box[2037] := 0.0;
   weight_box[2038] := 0.0;
   weight_box[2039] := 0.0;
   weight_box[2040] := 0.0;
   weight_box[2041] := 0.0;
   weight_box[2042] := 0.0;
   weight_box[2043] := 0.0;
   weight_box[2044] := 0.0;
   weight_box[2045] := 0.0;
   weight_box[2046] := 0.0;
   weight_box[2047] := 0.0;
   weight_box[2048] := 0.0;
   weight_box[2049] := 0.0;
   weight_box[2050] := 0.0;
   weight_box[2051] := 0.0;
   weight_box[2052] := 0.0;
   weight_box[2053] := 0.0;
   weight_box[2054] := 0.0;
   weight_box[2055] := 0.0;
   weight_box[2056] := 0.0;
   weight_box[2057] := 0.0;
   weight_box[2058] := 0.0;
   weight_box[2059] := 0.0;
   weight_box[2060] := 0.0;
   weight_box[2061] := 0.0;
   weight_box[2062] := 0.0;
   weight_box[2063] := 0.0;
   weight_box[2064] := 0.0;
   weight_box[2065] := 0.0;
   weight_box[2066] := 0.0;
   weight_box[2067] := 0.0;
   weight_box[2068] := 0.0;
   weight_box[2069] := 0.0;
   weight_box[2070] := 0.0;
   weight_box[2071] := 0.0;
   weight_box[2072] := 0.0;
   weight_box[2073] := 0.0;
   weight_box[2074] := 0.0;
   weight_box[2075] := 0.0;
   weight_box[2076] := 0.0;
   weight_box[2077] := 0.0;
   weight_box[2078] := 0.0;
   weight_box[2079] := 0.0;
   weight_box[2080] := 0.0;
   weight_box[2081] := 0.0;
   weight_box[2082] := 0.0;
   weight_box[2083] := 0.0;
   weight_box[2084] := 0.0;
   weight_box[2085] := 0.0;
   weight_box[2086] := 0.0;
   weight_box[2087] := 0.0;
   weight_box[2088] := 0.0;
   weight_box[2089] := 0.0;
   weight_box[2090] := 0.0;
   weight_box[2091] := 0.0;
   weight_box[2092] := 0.0;
   weight_box[2093] := 0.0;
   weight_box[2094] := 0.0;
   weight_box[2095] := 0.0;
   weight_box[2096] := 0.0;
   weight_box[2097] := 0.0;
   weight_box[2098] := 0.0;
   weight_box[2099] := 0.0;
   weight_box[2100] := 0.0;
   weight_box[2101] := 0.0;
   weight_box[2102] := 0.0;
   weight_box[2103] := 0.0;
   weight_box[2104] := 0.0;
   weight_box[2105] := 0.0;
   weight_box[2106] := 0.0;
   weight_box[2107] := 0.0;
   weight_box[2108] := 0.0;
   weight_box[2109] := 0.0;
   weight_box[2110] := 0.0;
   weight_box[2111] := 0.0;
   weight_box[2112] := 0.0;
   weight_box[2113] := 0.0;
   weight_box[2114] := 0.0;
   weight_box[2115] := 0.0;
   weight_box[2116] := 0.0;
   weight_box[2117] := 0.0;
   weight_box[2118] := 0.0;
   weight_box[2119] := 0.0;
   weight_box[2120] := 0.0;
   weight_box[2121] := 0.0;
   weight_box[2122] := 0.0;
   weight_box[2123] := 0.0;
   weight_box[2124] := 0.0;
   weight_box[2125] := 0.0;
   weight_box[2126] := 0.0;
   weight_box[2127] := 0.0;
   weight_box[2128] := 0.0;
   weight_box[2129] := 0.0;
   weight_box[2130] := 0.0;
   weight_box[2131] := 0.0;
   weight_box[2132] := 0.0;
   weight_box[2133] := 0.0;
   weight_box[2134] := 0.0;
   weight_box[2135] := 0.0;
   weight_box[2136] := 0.0;
   weight_box[2137] := 0.0;
   weight_box[2138] := 0.0;
   weight_box[2139] := 0.0;
   weight_box[2140] := 0.0;
   weight_box[2141] := 0.0;
   weight_box[2142] := 0.0;
   weight_box[2143] := 0.0;
   weight_box[2144] := 0.0;
   weight_box[2145] := 0.0;
   weight_box[2146] := 0.0;
   weight_box[2147] := 0.0;
   weight_box[2148] := 0.0;
   weight_box[2149] := 0.0;
   weight_box[2150] := 0.0;
   weight_box[2151] := 0.0;
   weight_box[2152] := 0.0;
   weight_box[2153] := 0.0;
   weight_box[2154] := 0.0;
   weight_box[2155] := 0.0;
   weight_box[2156] := 0.0;
   weight_box[2157] := 0.0;
   weight_box[2158] := 0.0;
   weight_box[2159] := 0.0;
   weight_box[2160] := 0.0;
   weight_box[2161] := 0.0;
   weight_box[2162] := 0.0;
   weight_box[2163] := 0.0;
   weight_box[2164] := 0.0;
   weight_box[2165] := 0.0;
   weight_box[2166] := 0.0;
   weight_box[2167] := 0.0;
   weight_box[2168] := 0.0;
   weight_box[2169] := 0.0;
   weight_box[2170] := 0.0;
   weight_box[2171] := 0.0;
   weight_box[2172] := 0.0;
   weight_box[2173] := 0.0;
   weight_box[2174] := 0.0;
   weight_box[2175] := 0.0;
   weight_box[2176] := 0.0;
   weight_box[2177] := 0.0;
   weight_box[2178] := 0.0;
   weight_box[2179] := 0.0;
   weight_box[2180] := 0.0;
   weight_box[2181] := 0.0;
   weight_box[2182] := 0.0;
   weight_box[2183] := 0.0;
   weight_box[2184] := 0.0;
   weight_box[2185] := 0.0;
   weight_box[2186] := 0.0;
   weight_box[2187] := 0.0;
   weight_box[2188] := 0.0;
   weight_box[2189] := 0.0;
   weight_box[2190] := 0.0;
   weight_box[2191] := 0.0;
   weight_box[2192] := 0.0;
   weight_box[2193] := 0.0;
   weight_box[2194] := 0.0;
   weight_box[2195] := 0.0;
   weight_box[2196] := 0.0;
   weight_box[2197] := 0.0;
   weight_box[2198] := 0.0;
   weight_box[2199] := 0.0;
   weight_box[2200] := 0.0;
END_DATA_BLOCK

// folder: (top level)

FUNCTION_BLOCK "Profinet_FC280"   // FB1, LAD
{ S7_Optimized_Access := 'FALSE' }
VERSION : 0.1
   VAR_INPUT
      In_Status : Word;
      In_FB : Word;
   END_VAR
   VAR_OUTPUT
      Out_CMD : Word;
      Out_SP : Word;
   END_VAR
   VAR
      Status_W : Word;
      Status : Struct
         Ready : Bool;   // Готов к управлению
         QF : Bool;   // Готов к работе / нет аварий
         Enable : Bool;   // Активен
         Trip : Bool;
         "ON 2" : Bool;
         "ON 3" : Bool;
         "Start not possible" : Bool;   // Запуск не возможен
         Warning : Bool;   // Предупреждение
         "Speed reference reached" : Bool;   // Скорость достигнута
         "Bus control" : Bool;
         "Frequency limit ok" : Bool;   // Максимальная частота
         Running : Bool;   // В работе
         Stopped : Bool;   // Остановлен
         "Voltage exceeded" : Bool;   // Ошибка по напряжению
         "Torque exceeded" : Bool;   // Ошибка по моменту
         "Timer exceeded" : Bool;   // Ошибка по времени
      END_STRUCT;
      In_FB_DI : DInt;
      In_FB_Real : Real;
      FB : Real;
      Out_W : Word;
      CMD : Struct
         "No stop" : Bool;
         "No coast stop" : Bool;
         "No quick stop" : Bool;
         "No coasting" : Bool;
         Ramp : Bool;
         "Use ramp" : Bool;
         Start : Bool;   // Запуск
         "Reset fault" : Bool;
         "Jog 1 ON" : Bool;
         "Jog 2 ON" : Bool;
         "Data valid" : Bool;
         "Slow down" : Bool;
         "Catch up" : Bool;
         "Selection lsb" : Bool;
         "Selection msb" : Bool;
         Reversing : Bool;
      END_STRUCT;
      SP : Real;   // Уставка
      SP_R : Real;
      SP_DI : DInt;
   END_VAR
   VAR_TEMP   // added for the SCL form of the ladder/FBD networks
      _w1 : Bool;
   END_VAR
BEGIN

REGION Network 1
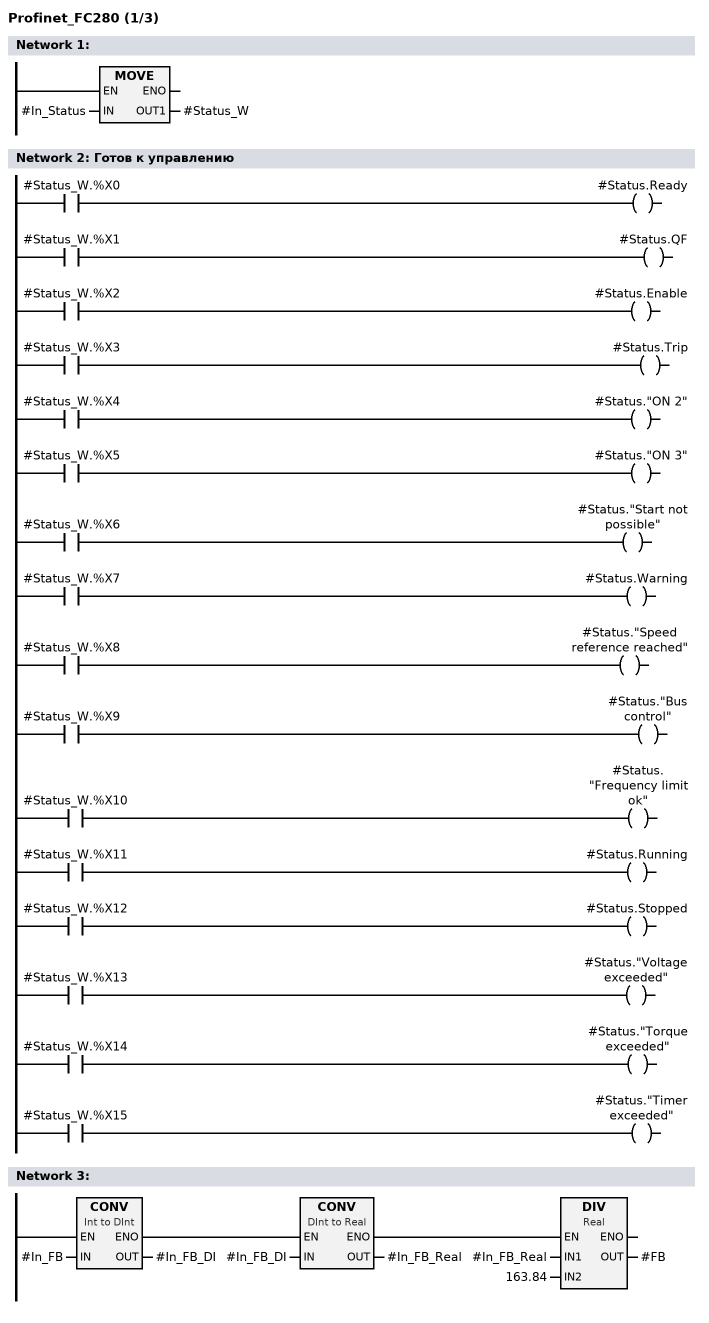
   RUNG wire#powerrail
      Move(in := #In_Status, out1 => #Status_W)
   END_RUNG
   // the same network as SCL:
   #Status_W := #In_Status;
END_REGION

REGION Network 2: Готов к управлению
   RUNG wire#powerrail
      Contact( #Status_W.%X0 )
      Coil( #Status.Ready )
   END_RUNG
   RUNG wire#powerrail
      Contact( #Status_W.%X1 )
      Coil( #Status.QF )
   END_RUNG
   RUNG wire#powerrail
      Contact( #Status_W.%X2 )
      Coil( #Status.Enable )
   END_RUNG
   RUNG wire#powerrail
      Contact( #Status_W.%X3 )
      Coil( #Status.Trip )
   END_RUNG
   RUNG wire#powerrail
      Contact( #Status_W.%X4 )
      Coil( #Status."ON 2" )
   END_RUNG
   RUNG wire#powerrail
      Contact( #Status_W.%X5 )
      Coil( #Status."ON 3" )
   END_RUNG
   RUNG wire#powerrail
      Contact( #Status_W.%X6 )
      Coil( #Status."Start not possible" )
   END_RUNG
   RUNG wire#powerrail
      Contact( #Status_W.%X7 )
      Coil( #Status.Warning )
   END_RUNG
   RUNG wire#powerrail
      Contact( #Status_W.%X8 )
      Coil( #Status."Speed reference reached" )
   END_RUNG
   RUNG wire#powerrail
      Contact( #Status_W.%X9 )
      Coil( #Status."Bus control" )
   END_RUNG
   RUNG wire#powerrail
      Contact( #Status_W.%X10 )
      Coil( #Status."Frequency limit ok" )
   END_RUNG
   RUNG wire#powerrail
      Contact( #Status_W.%X11 )
      Coil( #Status.Running )
   END_RUNG
   RUNG wire#powerrail
      Contact( #Status_W.%X12 )
      Coil( #Status.Stopped )
   END_RUNG
   RUNG wire#powerrail
      Contact( #Status_W.%X13 )
      Coil( #Status."Voltage exceeded" )
   END_RUNG
   RUNG wire#powerrail
      Contact( #Status_W.%X14 )
      Coil( #Status."Torque exceeded" )
   END_RUNG
   RUNG wire#powerrail
      Contact( #Status_W.%X15 )
      Coil( #Status."Timer exceeded" )
   END_RUNG
   // the same network as SCL:
   #Status.Ready := #Status_W.%X0;
   #Status.QF := #Status_W.%X1;
   #Status.Enable := #Status_W.%X2;
   #Status.Trip := #Status_W.%X3;
   #Status."ON 2" := #Status_W.%X4;
   #Status."ON 3" := #Status_W.%X5;
   #Status."Start not possible" := #Status_W.%X6;
   #Status.Warning := #Status_W.%X7;
   #Status."Speed reference reached" := #Status_W.%X8;
   #Status."Bus control" := #Status_W.%X9;
   #Status."Frequency limit ok" := #Status_W.%X10;
   #Status.Running := #Status_W.%X11;
   #Status.Stopped := #Status_W.%X12;
   #Status."Voltage exceeded" := #Status_W.%X13;
   #Status."Torque exceeded" := #Status_W.%X14;
   #Status."Timer exceeded" := #Status_W.%X15;
END_REGION

REGION Network 3
   RUNG wire#powerrail
      { S7_Templates := "[SrcType := Int, DestType := DInt]" } Convert(in := #In_FB, out => #In_FB_DI)
      { S7_Templates := "[SrcType := DInt, DestType := Real]" } Convert(in := #In_FB_DI, out => #In_FB_Real)
      { S7_Templates := "SrcType := Real" } Div(in1 := #In_FB_Real, in2 := 163.84, out => #FB)
   END_RUNG
   // the same network as SCL:
   #In_FB_DI := INT_TO_DINT(#In_FB);
   #In_FB_Real := DINT_TO_REAL(#In_FB_DI);
   #FB := #In_FB_Real / 163.84;
END_REGION

REGION Network 4
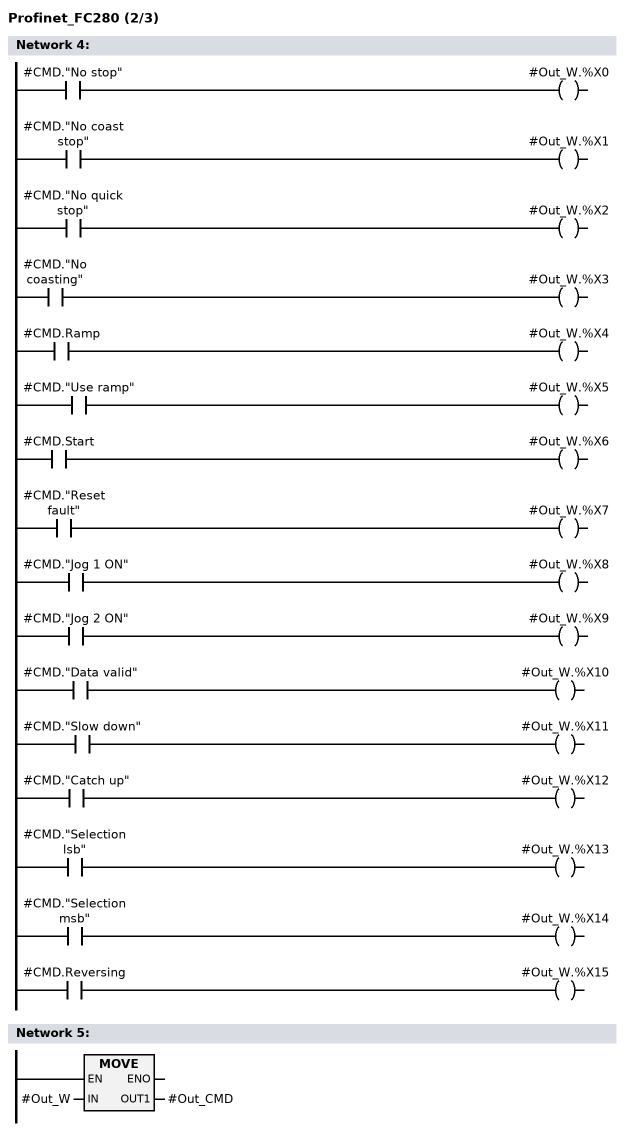
   RUNG wire#powerrail
      Contact( #CMD."No stop" )
      Coil( #Out_W.%X0 )
   END_RUNG
   RUNG wire#powerrail
      Contact( #CMD."No coast stop" )
      Coil( #Out_W.%X1 )
   END_RUNG
   RUNG wire#powerrail
      Contact( #CMD."No quick stop" )
      Coil( #Out_W.%X2 )
   END_RUNG
   RUNG wire#powerrail
      Contact( #CMD."No coasting" )
      Coil( #Out_W.%X3 )
   END_RUNG
   RUNG wire#powerrail
      Contact( #CMD.Ramp )
      Coil( #Out_W.%X4 )
   END_RUNG
   RUNG wire#powerrail
      Contact( #CMD."Use ramp" )
      Coil( #Out_W.%X5 )
   END_RUNG
   RUNG wire#powerrail
      Contact( #CMD.Start )
      Coil( #Out_W.%X6 )
   END_RUNG
   RUNG wire#powerrail
      Contact( #CMD."Reset fault" )
      Coil( #Out_W.%X7 )
   END_RUNG
   RUNG wire#powerrail
      Contact( #CMD."Jog 1 ON" )
      Coil( #Out_W.%X8 )
   END_RUNG
   RUNG wire#powerrail
      Contact( #CMD."Jog 2 ON" )
      Coil( #Out_W.%X9 )
   END_RUNG
   RUNG wire#powerrail
      Contact( #CMD."Data valid" )
      Coil( #Out_W.%X10 )
   END_RUNG
   RUNG wire#powerrail
      Contact( #CMD."Slow down" )
      Coil( #Out_W.%X11 )
   END_RUNG
   RUNG wire#powerrail
      Contact( #CMD."Catch up" )
      Coil( #Out_W.%X12 )
   END_RUNG
   RUNG wire#powerrail
      Contact( #CMD."Selection lsb" )
      Coil( #Out_W.%X13 )
   END_RUNG
   RUNG wire#powerrail
      Contact( #CMD."Selection msb" )
      Coil( #Out_W.%X14 )
   END_RUNG
   RUNG wire#powerrail
      Contact( #CMD.Reversing )
      Coil( #Out_W.%X15 )
   END_RUNG
   // the same network as SCL:
   #Out_W.%X0 := #CMD."No stop";
   #Out_W.%X1 := #CMD."No coast stop";
   #Out_W.%X2 := #CMD."No quick stop";
   #Out_W.%X3 := #CMD."No coasting";
   #Out_W.%X4 := #CMD.Ramp;
   #Out_W.%X5 := #CMD."Use ramp";
   #Out_W.%X6 := #CMD.Start;
   #Out_W.%X7 := #CMD."Reset fault";
   #Out_W.%X8 := #CMD."Jog 1 ON";
   #Out_W.%X9 := #CMD."Jog 2 ON";
   #Out_W.%X10 := #CMD."Data valid";
   #Out_W.%X11 := #CMD."Slow down";
   #Out_W.%X12 := #CMD."Catch up";
   #Out_W.%X13 := #CMD."Selection lsb";
   #Out_W.%X14 := #CMD."Selection msb";
   #Out_W.%X15 := #CMD.Reversing;
END_REGION

REGION Network 5
   RUNG wire#powerrail
      Move(in := #Out_W, out1 => #Out_CMD)
   END_RUNG
   // the same network as SCL:
   #Out_CMD := #Out_W;
END_REGION

REGION Network 6
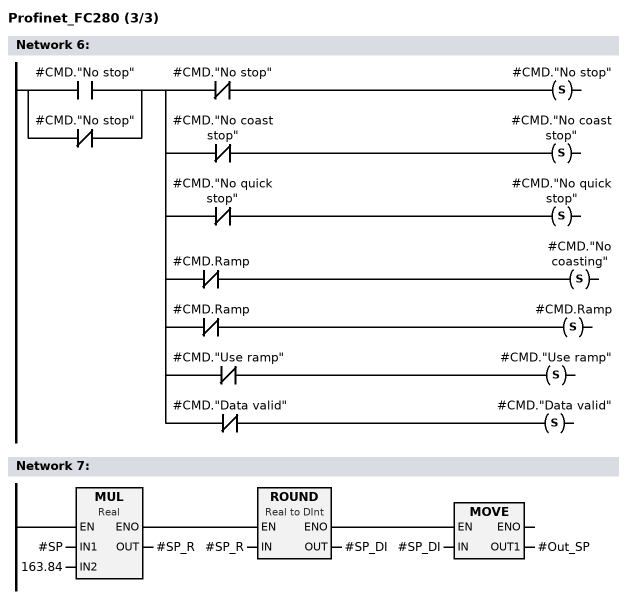
   RUNG wire#powerrail
      Contact( #CMD."No stop" )
      wire#w1
      I_Contact( #CMD."No stop" )
      S_Coil( #CMD."No stop" )
   END_RUNG
   RUNG wire#powerrail
      I_Contact( #CMD."No stop" )
   END_RUNG wire#w1
   RUNG wire#w1
      I_Contact( #CMD."No coast stop" )
      S_Coil( #CMD."No coast stop" )
   END_RUNG
   RUNG wire#w1
      I_Contact( #CMD."No quick stop" )
      S_Coil( #CMD."No quick stop" )
   END_RUNG
   RUNG wire#w1
      I_Contact( #CMD.Ramp )
      S_Coil( #CMD."No coasting" )
   END_RUNG
   RUNG wire#w1
      I_Contact( #CMD.Ramp )
      S_Coil( #CMD.Ramp )
   END_RUNG
   RUNG wire#w1
      I_Contact( #CMD."Use ramp" )
      S_Coil( #CMD."Use ramp" )
   END_RUNG
   RUNG wire#w1
      I_Contact( #CMD."Data valid" )
      S_Coil( #CMD."Data valid" )
   END_RUNG
   // the same network as SCL:
   #_w1 := #CMD."No stop" OR NOT #CMD."No stop";
   IF #_w1 AND NOT #CMD."No stop" THEN #CMD."No stop" := TRUE; END_IF;
   IF #_w1 AND NOT #CMD."No coast stop" THEN #CMD."No coast stop" := TRUE; END_IF;
   IF #_w1 AND NOT #CMD."No quick stop" THEN #CMD."No quick stop" := TRUE; END_IF;
   IF #_w1 AND NOT #CMD.Ramp THEN
       #CMD."No coasting" := TRUE;
       #CMD.Ramp := TRUE;
   END_IF;
   IF #_w1 AND NOT #CMD."Use ramp" THEN #CMD."Use ramp" := TRUE; END_IF;
   IF #_w1 AND NOT #CMD."Data valid" THEN #CMD."Data valid" := TRUE; END_IF;
END_REGION

REGION Network 7
   RUNG wire#powerrail
      { S7_Templates := "SrcType := Real" } Mul(in1 := #SP, in2 := 163.84, out => #SP_R)
      { S7_Templates := "[SrcType := Real, DestType := DInt]" } Round(in := #SP_R, out => #SP_DI)
      Move(in := #SP_DI, out1 => #Out_SP)
   END_RUNG
   // the same network as SCL:
   #SP_R := #SP * 163.84;
   #SP_DI := ROUND(#SP_R);
   #Out_SP := #SP_DI;
END_REGION
END_FUNCTION_BLOCK

FUNCTION_BLOCK "DRV_CF"   // FB4, LAD
{ S7_Optimized_Access := 'FALSE' }
VERSION : 0.1
   VAR_INPUT
      Start : Bool;   // Включить двигатель
      Coasting : Bool;   // СТОП ПЧ - свободный пробег
      Quick_stop : Bool;   // СТОП ПЧ - быстрый останов
      Kwit_alrm : Bool;   // Квитировать аварии
      SP : Real;   // Уставка частотника в процентах
   END_VAR
   VAR_OUTPUT
      Freq : Real;   // Текущая сглаженная частота
      Current : Real;   // Текущий ток нагруки
      Voltage : Real;   // Напряжение на выходе ПЧ
      Power : Real;   // Мощность
      Alarm : DWord;   // Код аварии
      Voltage_on_CF : Bool;   // Есть напряжение на ПЧ
      Alrm : Bool;   // Ошибка
      Warning : Bool;   // Предупреждение
      Ready_to_start : Bool;   // Готов к включению
      ON : Bool;   // Привод работает
      Relation_ok : Bool;   // Есть связь с частотником
   END_VAR
   VAR
      Status_Recive : Bool;   // Нормальный прием данных
      Status_Send : Bool;   // Нормальная передача данных
      Setbit : Bool;
      Error_Recive : Int;   // Код ошибки приема
      Error_Send : Int;   // Код ошибки передачи
      TMP_DI_1 : DInt;   // темп
      TMP_R_1 : Real;   // темп
      TMP_R_2 : Real;   // темп
      TMP_DI_2 : Real;   // темп
      TMP_R_3 : Real;   // темп
      TMP_DI_3 : DInt;   // темп
      TMP_R_4 : Real;   // темп
      TMP_R_5 : Real;   // темп
      TMP_DI_4 : Real;   // темп
      TMP_R_6 : Real;   // темп
      TMP_DI_5 : Real;   // темп
      TMP_DI_6 : DInt;   // темп
      Telegramm_input : Struct
         DEVIATION_SETPOINT : Bool;   // БИТ 08 Рассогласование уставки и фактического значения
         ASU_WORK : Bool;   // БИТ 09 Управление AG(PZD)
         MAX_FREQUENCY : Bool;   // БИТ 10 Достигнута максимальная частота
         PRIVOD_V_RABOTE : Bool;   // БИТ 11 Привод в работе
         RESERVED_12 : Bool;   // БИТ 12Не исп
         OVERLOAD_V : Bool;   // БИТ 13 Перегрузка по напряжению
         OVERLOAD_TORQUE : Bool;   // БИТ 14 Перегрузка по моменту
         THERMAL_WARNING : Bool;   // БИТ 15 Перегрев
         GOTOV_K_VKL : Bool;   // БИТ 00 Готов к включению
         GOTOV_K_RABOTE : Bool;   // БИТ 01 Готор к работе
         MOTOR_COASTING : Bool;   // БИТ 02 Останов с самовыбегом
         ALARM_ACTUAL : Bool;   // БИТ 03 Неисправность
         STOP2_PRIVOD : Bool;   // БИТ 04 ВЫКЛ 2
         STOP3_PRIVOD : Bool;   // БИТ 05 ВЫКЛ 3
         PUSK : Bool;   // БИТ 06 Есть команда старт
         WARNING_ACTUAL : Bool;   // БИТ 07 Предупреждение активно
         FREQUENCY : Word;   // Текущая частота
         CURRENT : DWord;   // Текущий ток
         VOLTAGE_MOTOR : Word;   // Напряжение на выходе
         VOLTAGE_DC : Word;   // Напряжение внутреннего контура
         POWER : DWord;   // Мощность
         ALARMS_CODES : DWord;   // Коды Аварий
      END_STRUCT;
      Telegramm_output : Struct
         JOG10FF : Bool;   // БИТ 08 Толчок вправо
         JOG20FF : Bool;   // БИТ 09 Толчок влево
         ASU_UPRAVLINIE : Bool;   // БИТ 10 Управление от контроллера
         SLOW_DOWN : Bool;   // БИТ 11 Уменьшить задание
         CATCH_UP : Bool;   // БИТ 12 Нарастить задание
         LSB : Bool;   // БИТ 13 определение номера настроек
         MSB : Bool;   // БИТ 14 определение номера настроек
         REVERSE : Bool;   // БИТ 15 реверс
         ON1 : Bool;   // БИТ 00 Разрешение на работу
         ON2 : Bool;   // БИТ 01 Разрешение на работу
         ON3 : Bool;   // БИТ 02 Разрешение на работу
         ENABLE : Bool;   // БИТ 03 Разрешение на работу
         QUICK_STOP : Bool;   // БИТ 04 Разрешение на работу
         FREEZE : Bool;   // БИТ 05 Разрешение на работу
         START : Bool;   // БИТ 06 Пуск двигателя
         KVIT_ALARM : Bool;   // Бит 7 сбой
         PID_SETPOINT : Word;   // уставка
         RESERVED3 : Word;   // резерв
         RESERVED4 : Word;   // резерв
         RESERVED5 : Word;   // резерв
         RESERVED6 : Word;   // резерв
         RESERVED7 : Word;   // резерв
         RESERVED8 : Word;   // резерв
      END_STRUCT;
   END_VAR
BEGIN

REGION Network 1
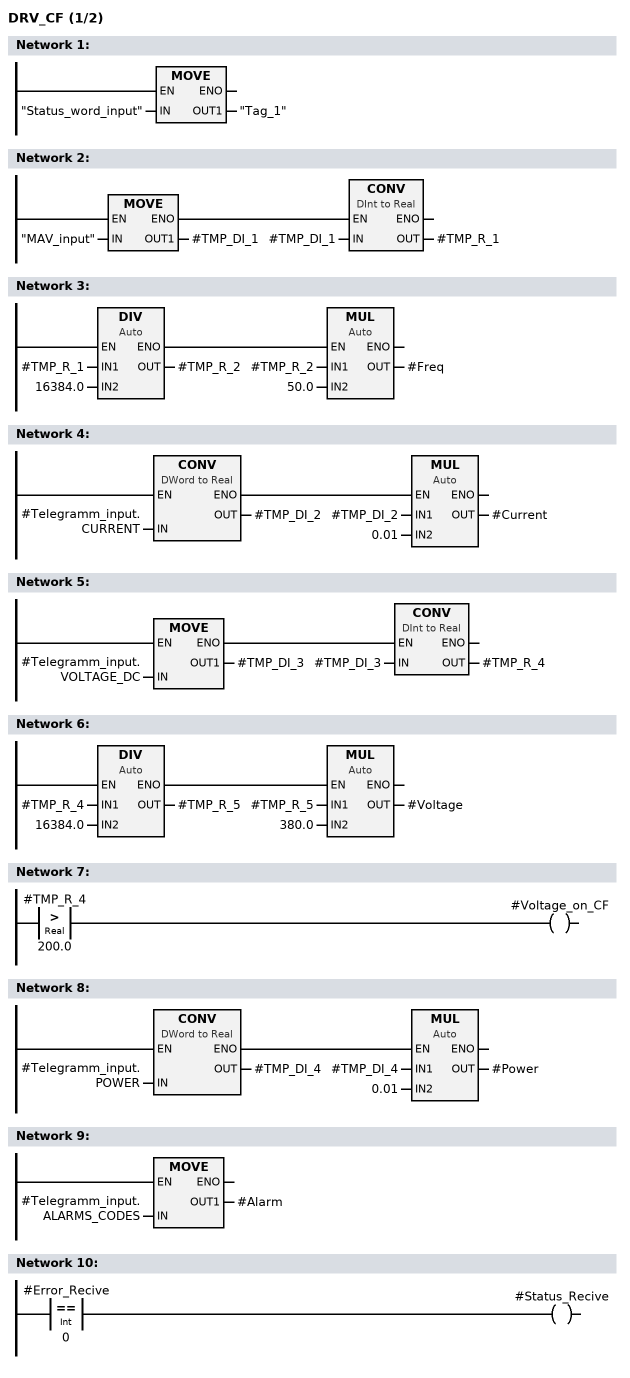
   RUNG wire#powerrail
      Move(in := "Status_word_input", out1 => "Tag_1")
   END_RUNG
   // the same network as SCL:
   "Tag_1" := "Status_word_input";
END_REGION

REGION Network 2
   RUNG wire#powerrail
      Move(in := "MAV_input", out1 => #TMP_DI_1)
      { S7_Templates := "[SrcType := DInt, DestType := Real]" } Convert(in := #TMP_DI_1, out => #TMP_R_1)
   END_RUNG
   // the same network as SCL:
   #TMP_DI_1 := "MAV_input";
   #TMP_R_1 := DINT_TO_REAL(#TMP_DI_1);
END_REGION

REGION Network 3
   RUNG wire#powerrail
      Div(in1 := #TMP_R_1, in2 := 16384.0, out => #TMP_R_2)
      Mul(in1 := #TMP_R_2, in2 := 50.0, out => #Freq)
   END_RUNG
   // the same network as SCL:
   #TMP_R_2 := #TMP_R_1 / 16384.0;
   #Freq := #TMP_R_2 * 50.0;
END_REGION

REGION Network 4
   RUNG wire#powerrail
      { S7_Templates := "[SrcType := DWord, DestType := Real]" } Convert(in := #Telegramm_input.CURRENT, out => #TMP_DI_2)
      Mul(in1 := #TMP_DI_2, in2 := 0.01, out => #Current)
   END_RUNG
   // the same network as SCL:
   #TMP_DI_2 := DWORD_TO_REAL(#Telegramm_input.CURRENT);
   #Current := #TMP_DI_2 * 0.01;
END_REGION

REGION Network 5
   RUNG wire#powerrail
      Move(in := #Telegramm_input.VOLTAGE_DC, out1 => #TMP_DI_3)
      { S7_Templates := "[SrcType := DInt, DestType := Real]" } Convert(in := #TMP_DI_3, out => #TMP_R_4)
   END_RUNG
   // the same network as SCL:
   #TMP_DI_3 := #Telegramm_input.VOLTAGE_DC;
   #TMP_R_4 := DINT_TO_REAL(#TMP_DI_3);
END_REGION

REGION Network 6
   RUNG wire#powerrail
      Div(in1 := #TMP_R_4, in2 := 16384.0, out => #TMP_R_5)
      Mul(in1 := #TMP_R_5, in2 := 380.0, out => #Voltage)
   END_RUNG
   // the same network as SCL:
   #TMP_R_5 := #TMP_R_4 / 16384.0;
   #Voltage := #TMP_R_5 * 380.0;
END_REGION

REGION Network 7
   RUNG wire#powerrail
      { S7_Templates := "SrcType := Real" } GT_Contact(in1 := #TMP_R_4, in2 := 200.0)
      Coil( #Voltage_on_CF )
   END_RUNG
   // the same network as SCL:
   #Voltage_on_CF := #TMP_R_4 > 200.0;
END_REGION

REGION Network 8
   RUNG wire#powerrail
      { S7_Templates := "[SrcType := DWord, DestType := Real]" } Convert(in := #Telegramm_input.POWER, out => #TMP_DI_4)
      Mul(in1 := #TMP_DI_4, in2 := 0.01, out => #Power)
   END_RUNG
   // the same network as SCL:
   #TMP_DI_4 := DWORD_TO_REAL(#Telegramm_input.POWER);
   #Power := #TMP_DI_4 * 0.01;
END_REGION

REGION Network 9
   RUNG wire#powerrail
      Move(in := #Telegramm_input.ALARMS_CODES, out1 => #Alarm)
   END_RUNG
   // the same network as SCL:
   #Alarm := #Telegramm_input.ALARMS_CODES;
END_REGION

REGION Network 10
   RUNG wire#powerrail
      { S7_Templates := "SrcType := Int" } EQ_Contact(in1 := #Error_Recive, in2 := 0)
      Coil( #Status_Recive )
   END_RUNG
   // the same network as SCL:
   #Status_Recive := #Error_Recive = 0;
END_REGION

REGION Network 11
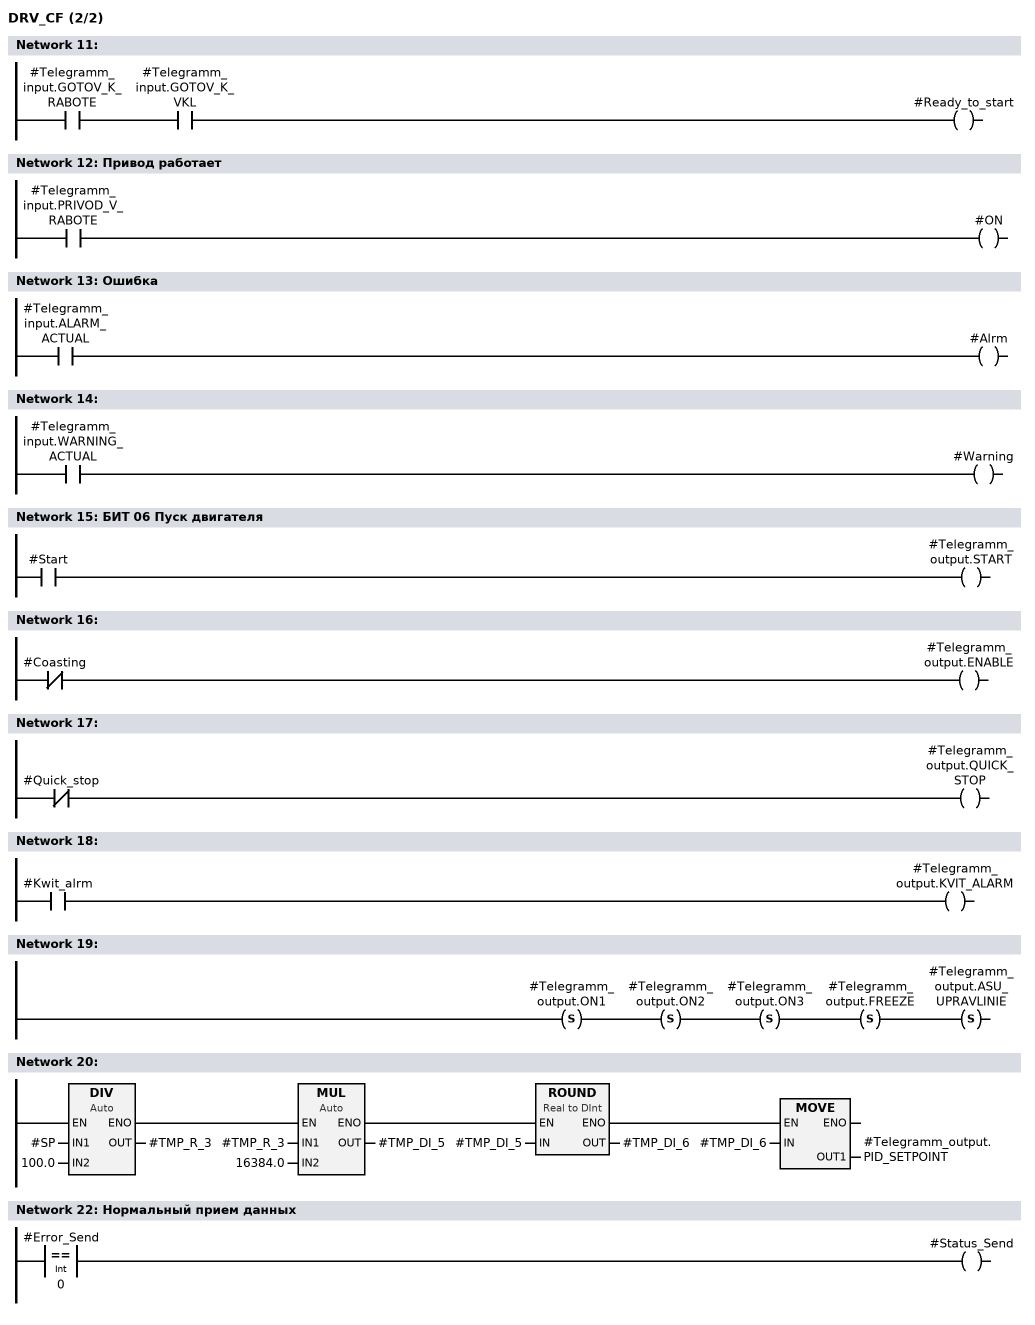
   RUNG wire#powerrail
      Contact( #Telegramm_input.GOTOV_K_RABOTE )
      Contact( #Telegramm_input.GOTOV_K_VKL )
      Coil( #Ready_to_start )
   END_RUNG
   // the same network as SCL:
   #Ready_to_start := #Telegramm_input.GOTOV_K_RABOTE AND #Telegramm_input.GOTOV_K_VKL;
END_REGION

REGION Network 12: Привод работает
   RUNG wire#powerrail
      Contact( #Telegramm_input.PRIVOD_V_RABOTE )
      Coil( #ON )
   END_RUNG
   // the same network as SCL:
   #ON := #Telegramm_input.PRIVOD_V_RABOTE;
END_REGION

REGION Network 13: Ошибка
   RUNG wire#powerrail
      Contact( #Telegramm_input.ALARM_ACTUAL )
      Coil( #Alrm )
   END_RUNG
   // the same network as SCL:
   #Alrm := #Telegramm_input.ALARM_ACTUAL;
END_REGION

REGION Network 14
   RUNG wire#powerrail
      Contact( #Telegramm_input.WARNING_ACTUAL )
      Coil( #Warning )
   END_RUNG
   // the same network as SCL:
   #Warning := #Telegramm_input.WARNING_ACTUAL;
END_REGION

REGION Network 15: БИТ 06 Пуск двигателя
   RUNG wire#powerrail
      Contact( #Start )
      Coil( #Telegramm_output.START )
   END_RUNG
   // the same network as SCL:
   #Telegramm_output.START := #Start;
END_REGION

REGION Network 16
   RUNG wire#powerrail
      I_Contact( #Coasting )
      Coil( #Telegramm_output.ENABLE )
   END_RUNG
   // the same network as SCL:
   #Telegramm_output.ENABLE := NOT #Coasting;
END_REGION

REGION Network 17
   RUNG wire#powerrail
      I_Contact( #Quick_stop )
      Coil( #Telegramm_output.QUICK_STOP )
   END_RUNG
   // the same network as SCL:
   #Telegramm_output.QUICK_STOP := NOT #Quick_stop;
END_REGION

REGION Network 18
   RUNG wire#powerrail
      Contact( #Kwit_alrm )
      Coil( #Telegramm_output.KVIT_ALARM )
   END_RUNG
   // the same network as SCL:
   #Telegramm_output.KVIT_ALARM := #Kwit_alrm;
END_REGION

REGION Network 19
   RUNG wire#powerrail
      S_Coil( #Telegramm_output.ON1 )
      S_Coil( #Telegramm_output.ON2 )
      S_Coil( #Telegramm_output.ON3 )
      S_Coil( #Telegramm_output.FREEZE )
      S_Coil( #Telegramm_output.ASU_UPRAVLINIE )
   END_RUNG
   // the same network as SCL:
   #Telegramm_output.ON1 := TRUE;
   #Telegramm_output.ON2 := TRUE;
   #Telegramm_output.ON3 := TRUE;
   #Telegramm_output.FREEZE := TRUE;
   #Telegramm_output.ASU_UPRAVLINIE := TRUE;
END_REGION

REGION Network 20
   RUNG wire#powerrail
      Div(in1 := #SP, in2 := 100.0, out => #TMP_R_3)
      Mul(in1 := #TMP_R_3, in2 := 16384.0, out => #TMP_DI_5)
      { S7_Templates := "[SrcType := Real, DestType := DInt]" } Round(in := #TMP_DI_5, out => #TMP_DI_6)
      Move(in := #TMP_DI_6, out1 => #Telegramm_output.PID_SETPOINT)
   END_RUNG
   // the same network as SCL:
   #TMP_R_3 := #SP / 100.0;
   #TMP_DI_5 := #TMP_R_3 * 16384.0;
   #TMP_DI_6 := ROUND(#TMP_DI_5);
   #Telegramm_output.PID_SETPOINT := #TMP_DI_6;
END_REGION

REGION Network 22: Нормальный прием данных
   RUNG wire#powerrail
      { S7_Templates := "SrcType := Int" } EQ_Contact(in1 := #Error_Send, in2 := 0)
      Coil( #Status_Send )
   END_RUNG
   // the same network as SCL:
   #Status_Send := #Error_Send = 0;
END_REGION
END_FUNCTION_BLOCK

FUNCTION_BLOCK "T4D4"   // FB5, LAD
TITLE = Управление транспортером 4
{ S7_Optimized_Access := 'FALSE' }
VERSION : 0.1
   VAR_INPUT
      Start_weight : Bool;
      D4 : Bool;
      Alarm : Bool;
   END_VAR
   VAR_OUTPUT
      Ready : Bool;
      CMD_T4 : Bool;
   END_VAR
   VAR
      S1 : Struct
         SP : Real;   // Уставка
         Now : Real;   // Текущий счёт
         One : Real;   // Вес импульса
         Progress : Real;   // Прогресс выполнения
         "Exit" : Bool;   // Счёт завершён
         Start : Bool;   // Запуск
         Pause : Bool;   // Пауза
         Reset : Bool;   // Сброс счёта
         pos : Bool;   // Контроль фронта сигнала
      END_STRUCT;
      "Step" : Int;
      S2 : Struct
         SP : Real;   // Уставка
         Now : Real;   // Текущий счёт
         One : Real;   // Вес импульса
         Progress : Real;   // Прогресс выполнения
         "Exit" : Bool;   // Счёт завершён
         Start : Bool;   // Запуск
         Pause : Bool;   // Пауза
         Reset : Bool;   // Сброс счёта
         pos : Bool;   // Контроль фронта сигнала
      END_STRUCT;
   END_VAR
   VAR_TEMP   // added for the SCL form of the ladder/FBD networks
      _w1 : Bool;
   END_VAR
BEGIN

REGION Network 1: нет вкл - нулевой шаг, транспортер стоит
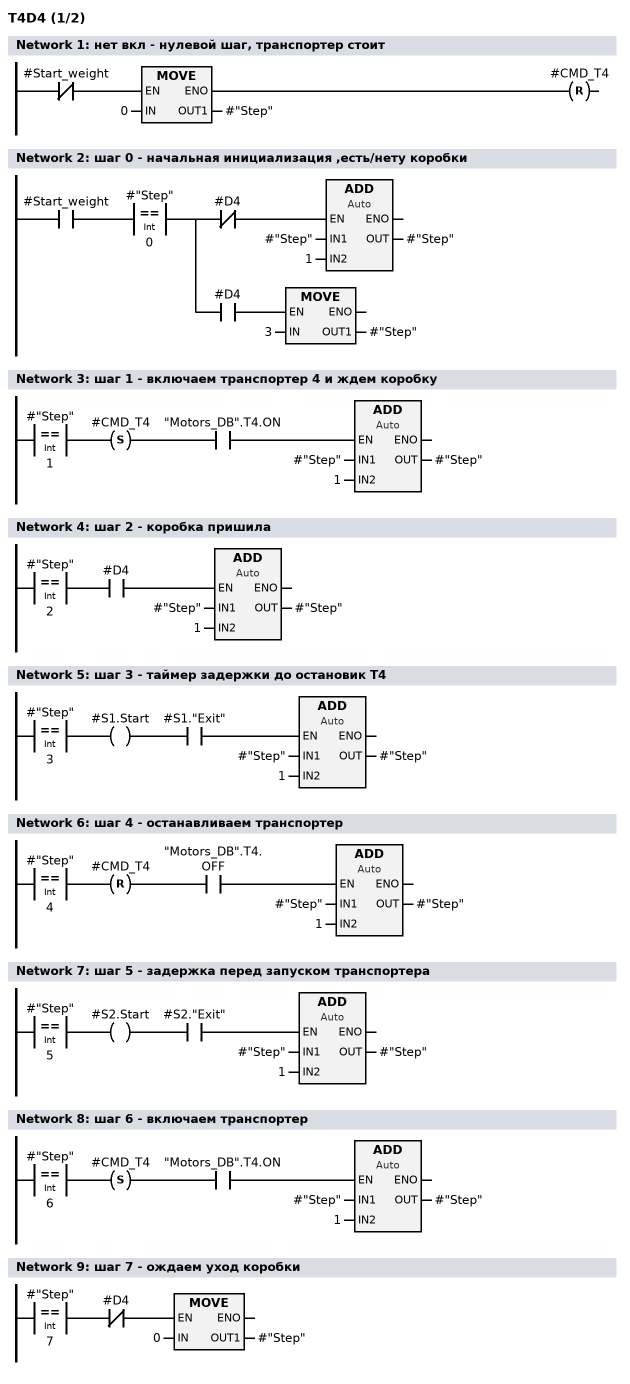
   RUNG wire#powerrail
      I_Contact( #Start_weight )
      Move(in := 0, out1 => #"Step")
      R_Coil( #CMD_T4 )
   END_RUNG
   // the same network as SCL:
   IF NOT #Start_weight THEN
       #"Step" := 0;
       #CMD_T4 := FALSE;
   END_IF;
END_REGION

REGION Network 2: шаг 0 - начальная инициализация ,есть/нету коробки
   RUNG wire#powerrail
      Contact( #Start_weight )
      { S7_Templates := "SrcType := Int" } EQ_Contact(in1 := #"Step", in2 := 0)
      wire#w1
      I_Contact( #D4 )
      Add(in1 := #"Step", in2 := 1, out => #"Step")
   END_RUNG
   RUNG wire#w1
      Contact( #D4 )
      Move(in := 3, out1 => #"Step")
   END_RUNG
   // the same network as SCL:
   #_w1 := #Start_weight AND (#"Step" = 0);
   IF #_w1 AND NOT #D4 THEN #"Step" := #"Step" + 1; END_IF;
   IF #_w1 AND #D4 THEN #"Step" := 3; END_IF;
END_REGION

REGION Network 3: шаг 1 - включаем транспортер 4 и ждем коробку
   RUNG wire#powerrail
      { S7_Templates := "SrcType := Int" } EQ_Contact(in1 := #"Step", in2 := 1)
      S_Coil( #CMD_T4 )
      Contact( "Motors_DB".T4.ON )
      Add(in1 := #"Step", in2 := 1, out => #"Step")
   END_RUNG
   // the same network as SCL:
   #_w1 := #"Step" = 1;
   IF #_w1 THEN #CMD_T4 := TRUE; END_IF;
   IF #_w1 AND "Motors_DB".T4.ON THEN #"Step" := #"Step" + 1; END_IF;
END_REGION

REGION Network 4: шаг 2 - коробка пришила
   RUNG wire#powerrail
      { S7_Templates := "SrcType := Int" } EQ_Contact(in1 := #"Step", in2 := 2)
      Contact( #D4 )
      Add(in1 := #"Step", in2 := 1, out => #"Step")
   END_RUNG
   // the same network as SCL:
   IF (#"Step" = 2) AND #D4 THEN #"Step" := #"Step" + 1; END_IF;
END_REGION

REGION Network 5: шаг 3 - таймер задержки до остановик Т4
   RUNG wire#powerrail
      { S7_Templates := "SrcType := Int" } EQ_Contact(in1 := #"Step", in2 := 3)
      Coil( #S1.Start )
      Contact( #S1."Exit" )
      Add(in1 := #"Step", in2 := 1, out => #"Step")
   END_RUNG
   // the same network as SCL:
   #S1.Start := #"Step" = 3;
   IF #S1.Start AND #S1."Exit" THEN #"Step" := #"Step" + 1; END_IF;
END_REGION

REGION Network 6: шаг 4 - останавливаем транспортер
   RUNG wire#powerrail
      { S7_Templates := "SrcType := Int" } EQ_Contact(in1 := #"Step", in2 := 4)
      R_Coil( #CMD_T4 )
      Contact( "Motors_DB".T4.OFF )
      Add(in1 := #"Step", in2 := 1, out => #"Step")
   END_RUNG
   // the same network as SCL:
   #_w1 := #"Step" = 4;
   IF #_w1 THEN #CMD_T4 := FALSE; END_IF;
   IF #_w1 AND "Motors_DB".T4.OFF THEN #"Step" := #"Step" + 1; END_IF;
END_REGION

REGION Network 7: шаг 5 - задержка перед запуском транспортера
   RUNG wire#powerrail
      { S7_Templates := "SrcType := Int" } EQ_Contact(in1 := #"Step", in2 := 5)
      Coil( #S2.Start )
      Contact( #S2."Exit" )
      Add(in1 := #"Step", in2 := 1, out => #"Step")
   END_RUNG
   // the same network as SCL:
   #S2.Start := #"Step" = 5;
   IF #S2.Start AND #S2."Exit" THEN #"Step" := #"Step" + 1; END_IF;
END_REGION

REGION Network 8: шаг 6 - включаем транспортер
   RUNG wire#powerrail
      { S7_Templates := "SrcType := Int" } EQ_Contact(in1 := #"Step", in2 := 6)
      S_Coil( #CMD_T4 )
      Contact( "Motors_DB".T4.ON )
      Add(in1 := #"Step", in2 := 1, out => #"Step")
   END_RUNG
   // the same network as SCL:
   #_w1 := #"Step" = 6;
   IF #_w1 THEN #CMD_T4 := TRUE; END_IF;
   IF #_w1 AND "Motors_DB".T4.ON THEN #"Step" := #"Step" + 1; END_IF;
END_REGION

REGION Network 9: шаг 7 - ождаем уход коробки
   RUNG wire#powerrail
      { S7_Templates := "SrcType := Int" } EQ_Contact(in1 := #"Step", in2 := 7)
      I_Contact( #D4 )
      Move(in := 0, out1 => #"Step")
   END_RUNG
   // the same network as SCL:
   IF (#"Step" = 7) AND NOT #D4 THEN #"Step" := 0; END_IF;
END_REGION

REGION Network 10: Готовность принять следующую коробку, если транспортер вкл и нет сигнала датчика
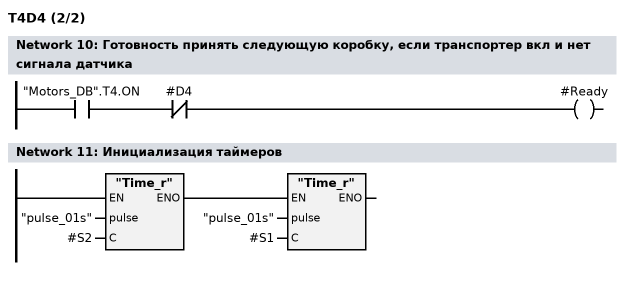
   RUNG wire#powerrail
      Contact( "Motors_DB".T4.ON )
      I_Contact( #D4 )
      Coil( #Ready )
   END_RUNG
   // the same network as SCL:
   #Ready := "Motors_DB".T4.ON AND NOT #D4;
END_REGION

REGION Network 11: Инициализация таймеров
   RUNG wire#powerrail
      "Time_r"(pulse := "pulse_01s", C := #S2)
      "Time_r"(pulse := "pulse_01s", C := #S1)
   END_RUNG
   // the same network as SCL:
   "Time_r"(pulse := "pulse_01s", C := #S2, ENO => #_w1);
   IF #_w1 THEN "Time_r"(pulse := "pulse_01s", C := #S1); END_IF;
END_REGION
END_FUNCTION_BLOCK

FUNCTION_BLOCK "Logic"   // FB6, LAD
{ S7_Optimized_Access := 'FALSE' }
VERSION : 0.1
   VAR
      DL : Struct
         stateMem_9 : Bool;
         stateMem_8 : Bool;
         stateMem_7 : Bool;
         stateMem_6 : Bool;
         stateMem_5 : Bool;
         stateMem_4 : Bool;
         stateMem_3 : Bool;
         stateMem_2 : Bool;
         stateMem_1 : Bool;
         stateMem : Bool;
      END_STRUCT;
      Clear_mem : Bool;
      proba : Struct
         i : Int := 1;
         x1 : Bool;
         x5 : Bool;
         x4 : Bool;
         x3 : Bool;
         x2 : Bool;
         pulse : Bool;
         null : DWord;
         "name" : String := 'del1';
      END_STRUCT;
      DataLogDelete_Instance_1 : DataLogDelete;
      count_block : Int;
      delet_block : String;
      x6 : Bool;
      x5 : Bool;
      x1 : Bool;
      x4 : Bool;
      x3 : Bool;
      x2 : Bool;
      crate_DL : Bool;
      Hand : Bool;
      stateMem : Bool;
      Start_weight : Bool;
      Alarm : Word;
      count : Int;
      "real" : Real;
      T_reset : Struct
         SP : Real := 1.0;   // Уставка
         Now : Real;   // Текущий счёт
         One : Real := 0.1;   // Вес импульса
         Progress : Real;   // Прогресс выполнения
         "Exit" : Bool;   // Счёт завершён
         Start : Bool;   // Запуск
         Pause : Bool;   // Пауза
         Reset : Bool;   // Сброс счёта
         pos : Bool;   // Контроль фронта сигнала
      END_STRUCT;
      T_reset_mem : Struct
         SP : Real := 1.0;   // Уставка
         Now : Real;   // Текущий счёт
         One : Real := 0.1;   // Вес импульса
         Progress : Real;   // Прогресс выполнения
         "Exit" : Bool;   // Счёт завершён
         Start : Bool;   // Запуск
         Pause : Bool;   // Пауза
         Reset : Bool;   // Сброс счёта
         pos : Bool;   // Контроль фронта сигнала
      END_STRUCT;
      DataLogCreate_Instance : DataLogCreate;
      DataLogWrite_Instance : DataLogWrite;
      DataLogClose_Instance : DataLogClose;
      DataLogOpen_Instance : DataLogOpen;
      DataLogNewFile_Instance : DataLogNewFile;
      DataLogClear_Instance : DataLogClear;
      DataLogDelete_Instance : DataLogDelete;
   END_VAR
   VAR_TEMP   // added for the SCL form of the ladder/FBD networks
      _w1 : Bool;
      _w2 : Bool;
   END_VAR
BEGIN

REGION Network 1: статистика
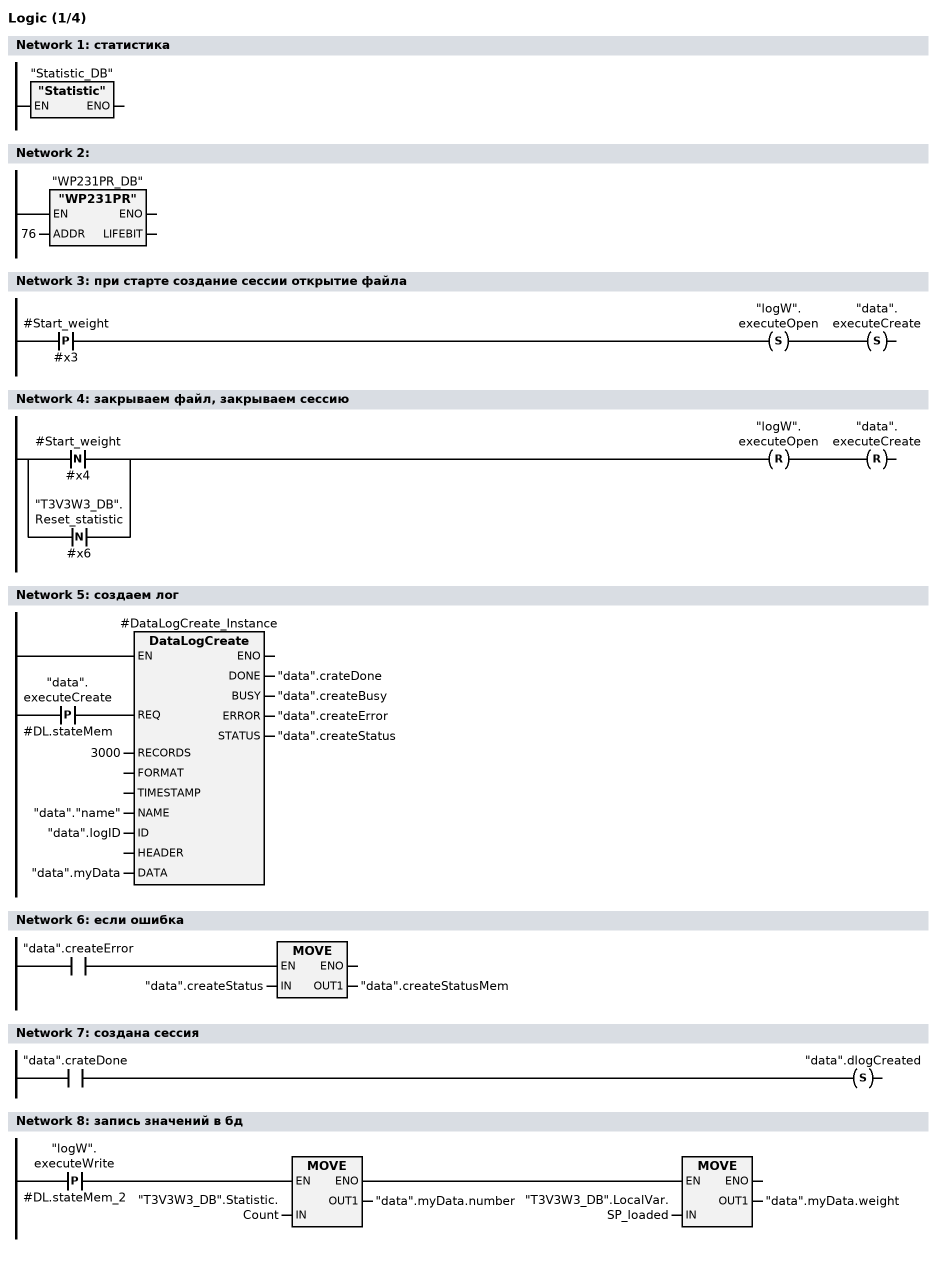
   RUNG wire#powerrail
      "Statistic_DB"()
   END_RUNG
   // the same network as SCL:
   "Statistic_DB"();   // "Statistic"
END_REGION

REGION Network 2
   RUNG wire#powerrail
      "WP231PR_DB"(ADDR := 76, LIFEBIT =>)
   END_RUNG
   // the same network as SCL:
   "WP231PR_DB"(ADDR := 76);   // "WP231PR"
END_REGION

REGION Network 3: при старте создание сессии открытие файла
   RUNG wire#powerrail
      P_Contact(operand := #Start_weight, bit := #x3)
      S_Coil( "logW".executeOpen )
      S_Coil( "data".executeCreate )
   END_RUNG
   // the same network as SCL:
   #_w1 := #Start_weight AND NOT #x3;   // rising edge of #Start_weight
   #x3 := #Start_weight;
   IF #_w1 THEN
       "logW".executeOpen := TRUE;
       "data".executeCreate := TRUE;
   END_IF;
END_REGION

REGION Network 4: закрываем файл, закрываем сессию
   RUNG wire#powerrail
      N_Contact(operand := #Start_weight, bit := #x4)
      wire#w1
      R_Coil( "logW".executeOpen )
      R_Coil( "data".executeCreate )
   END_RUNG
   RUNG wire#powerrail
      N_Contact(operand := "T3V3W3_DB".Reset_statistic, bit := #x6)
   END_RUNG wire#w1
   // the same network as SCL:
   #_w1 := NOT #Start_weight AND #x4;   // falling edge of #Start_weight
   #x4 := #Start_weight;
   #_w2 := NOT "T3V3W3_DB".Reset_statistic AND #x6;   // falling edge of "T3V3W3_DB".Reset_statistic
   #x6 := "T3V3W3_DB".Reset_statistic;
   IF #_w1 OR #_w2 THEN
       "logW".executeOpen := FALSE;
       "data".executeCreate := FALSE;
   END_IF;
END_REGION

